LIN {X 0,Y 195.024,Z 1205.929,A -85,B 0,C 180,E1 26196.812,E2 26196.812} C_VEL
LIN {X 0,Y 201.887,Z 1195.668,A -85,B 0,C 180,E1 26216.922,E2 26216.922} C_VEL
LIN {X 0,Y 228.615,Z 1170.249,A -85,B 0,C 180,E1 26237.028,E2 26237.028} C_VEL
LIN {X 0,Y 271.892,Z 1129.75,A -85,B 0,C 180,E1 26251.738,E2 26251.738} C_VEL
LIN {X 0,Y 319.813,Z 1076.72,A -85,B 0,C 180,E1 26261.083,E2 26261.083} C_VEL
LIN {X 0,Y 361.01,Z 1018.168,A -85,B 0,C 180,E1 26266.67,E2 26266.67} C_VEL
LIN {X 0,Y 361.601,Z 999.754,A -85,B 0,C 180,E1 26275.219,E2 26275.219} C_VEL
LIN {X 0,Y 361.684,Z 993.07,A -85,B 0,C 180,E1 26283.639,E2 26283.639} C_VEL
LIN {X 0,Y 360.895,Z 1000.649,A -85,B 0,C 180,E1 26292.409,E2 26292.409} C_VEL
LIN {X 0,Y 359.633,Z 1018.396,A -85,B 0,C 180,E1 26300.562,E2 26300.562} C_VEL
LIN {X 0,Y 315.236,Z 1080.357,A -85,B 0,C 180,E1 26306.923,E2 26306.923} C_VEL
LIN {X 0,Y 267.258,Z 1131.688,A -85,B 0,C 180,E1 26316.736,E2 26316.736} C_VEL
LIN {X 0,Y 264.551,Z 1134.275,A -85,B 0,C 180,E1 26317.455,E2 26317.455} C_VEL
LIN {X 0,Y 240.513,Z 1151.989,A -85,B 0,C 180,E1 26321.828,E2 26321.828} C_VEL
LIN {X 0,Y 204.312,Z 1182.961,A -85,B 0,C 180,E1 26339.909,E2 26339.909} C_VEL
LIN {X 0,Y 188.932,Z 1198.697,A -85,B 0,C 180,E1 26360.642,E2 26360.642} C_VEL
LIN {X 0,Y 186.458,Z 1202.773,A -85,B 0,C 180,E1 26376.895,E2 26376.895} C_VEL
LIN {X 0,Y 189.671,Z 1199.838,A -85,B 0,C 180,E1 26395.976,E2 26395.976} C_VEL
LIN {X 0,Y 209.352,Z 1185.393,A -85,B 0,C 180,E1 26417.213,E2 26417.213} C_VEL
LIN {X 0,Y 251.624,Z 1155.697,A -85,B 0,C 180,E1 26434.833,E2 26434.833} C_VEL
LIN {X 0,Y 304.449,Z 1112.39,A -85,B 0,C 180,E1 26446.069,E2 26446.069} C_VEL
LIN {X 0,Y 355.93,Z 1058.355,A -85,B 0,C 180,E1 26452.911,E2 26452.911} C_VEL
LIN {X 0,Y 371.692,Z 1038.15,A -85,B 0,C 180,E1 26454.701,E2 26454.701} C_VEL
LIN {X 0,Y 373.231,Z 1031.62,A -85,B 0,C 180,E1 26461.134,E2 26461.134} C_VEL
LIN {X 0,Y 372.915,Z 1033.797,A -85,B 0,C 180,E1 26468.154,E2 26468.154} C_VEL
LIN {X 0,Y 370.664,Z 1040.666,A -85,B 0,C 180,E1 26472.243,E2 26472.243} C_VEL
LIN {X 0,Y 321.62,Z 1097.337,A -85,B 0,C 180,E1 26477.917,E2 26477.917} C_VEL
LIN {X 0,Y 267.836,Z 1145.357,A -85,B 0,C 180,E1 26487.532,E2 26487.532} C_VEL
LIN {X 0,Y 221.377,Z 1179.857,A -85,B 0,C 180,E1 26502.685,E2 26502.685} C_VEL
LIN {X 0,Y 192.93,Z 1200.687,A -85,B 0,C 180,E1 26524.578,E2 26524.578} C_VEL
LIN {X 0,Y 187.059,Z 1206.716,A -85,B 0,C 180,E1 26543.127,E2 26543.127} C_VEL
LIN {X 0,Y 187.015,Z 1205.813,A -85,B 0,C 180,E1 26557.105,E2 26557.105} C_VEL
LIN {X 0,Y 194.537,Z 1195.482,A -85,B 0,C 180,E1 26578.027,E2 26578.027} C_VEL
LIN {X 0,Y 223.002,Z 1169.972,A -85,B 0,C 180,E1 26598.599,E2 26598.599} C_VEL
LIN {X 0,Y 268.014,Z 1129.339,A -85,B 0,C 180,E1 26613.321,E2 26613.321} C_VEL
LIN {X 0,Y 316.678,Z 1076.788,A -85,B 0,C 180,E1 26622.446,E2 26622.446} C_VEL
LIN {X 0,Y 356.066,Z 1022.174,A -85,B 0,C 180,E1 26627.651,E2 26627.651} C_VEL
LIN {X 0,Y 357.113,Z 1004.901,A -85,B 0,C 180,E1 26636.379,E2 26636.379} C_VEL
LIN {X 0,Y 357.474,Z 999.9,A -85,B 0,C 180,E1 26643.682,E2 26643.682} C_VEL
LIN {X 0,Y 356.208,Z 1008.216,A -85,B 0,C 180,E1 26652.952,E2 26652.952} C_VEL
LIN {X 0,Y 353.927,Z 1024.296,A -85,B 0,C 180,E1 26659.943,E2 26659.943} C_VEL
LIN {X 0,Y 308.648,Z 1084.424,A -85,B 0,C 180,E1 26666.084,E2 26666.084} C_VEL
LIN {X 0,Y 259.49,Z 1134.902,A -85,B 0,C 180,E1 26676.09,E2 26676.09} C_VEL
LIN {X 0,Y 240.513,Z 1151.989,A -85,B 0,C 180,E1 26681.828,E2 26681.828} C_VEL
LIN {X 0,Y 216.948,Z 1167.301,A -85,B 0,C 180,E1 26687.305,E2 26687.305} C_VEL
LIN {X 0,Y 187.065,Z 1192.104,A -85,B 0,C 180,E1 26708.47,E2 26708.47} C_VEL
LIN {X 0,Y 179.568,Z 1201.352,A -85,B 0,C 180,E1 26727.459,E2 26727.459} C_VEL
LIN {X 0,Y 178.358,Z 1202.913,A -85,B 0,C 180,E1 26742.156,E2 26742.156} C_VEL
LIN {X 0,Y 186.636,Z 1196.622,A -85,B 0,C 180,E1 26764.382,E2 26764.382} C_VEL
LIN {X 0,Y 218.438,Z 1175.736,A -85,B 0,C 180,E1 26786.538,E2 26786.538} C_VEL
LIN {X 0,Y 267.906,Z 1140.876,A -85,B 0,C 180,E1 26801.382,E2 26801.382} C_VEL
LIN {X 0,Y 323.344,Z 1092.416,A -85,B 0,C 180,E1 26810.602,E2 26810.602} C_VEL
LIN {X 0,Y 366.777,Z 1043.151,A -85,B 0,C 180,E1 26815.553,E2 26815.553} C_VEL
LIN {X 0,Y 368.312,Z 1037.517,A -85,B 0,C 180,E1 26823.511,E2 26823.511} C_VEL
LIN {X 0,Y 366.986,Z 1043.658,A -85,B 0,C 180,E1 26831.058,E2 26831.058} C_VEL
LIN {X 0,Y 314.684,Z 1102.026,A -85,B 0,C 180,E1 26837.109,E2 26837.109} C_VEL
LIN {X 0,Y 259.292,Z 1149.207,A -85,B 0,C 180,E1 26847.01,E2 26847.01} C_VEL
LIN {X 0,Y 210.752,Z 1183.326,A -85,B 0,C 180,E1 26863.433,E2 26863.433} C_VEL
LIN {X 0,Y 183.93,Z 1201.951,A -85,B 0,C 180,E1 26885.994,E2 26885.994} C_VEL
LIN {X 0,Y 178.992,Z 1206.922,A -85,B 0,C 180,E1 26907.691,E2 26907.691} C_VEL
LIN {X 0,Y 180.833,Z 1202.479,A -85,B 0,C 180,E1 26927.202,E2 26927.202} C_VEL
LIN {X 0,Y 197.975,Z 1185.627,A -85,B 0,C 180,E1 26949.358,E2 26949.358} C_VEL
LIN {X 0,Y 236.545,Z 1153.621,A -85,B 0,C 180,E1 26967.534,E2 26967.534} C_VEL
LIN {X 0,Y 286.12,Z 1107.52,A -85,B 0,C 180,E1 26979.377,E2 26979.377} C_VEL
LIN {X 0,Y 335.559,Z 1049.133,A -85,B 0,C 180,E1 26986.721,E2 26986.721} C_VEL
LIN {X 0,Y 351.217,Z 1025.839,A -85,B 0,C 180,E1 26988.826,E2 26988.826} C_VEL
LIN {X 0,Y 352.633,Z 1010,A -85,B 0,C 180,E1 26997.721,E2 26997.721} C_VEL
LIN {X 0,Y 352.974,Z 1006.543,A -85,B 0,C 180,E1 27003.729,E2 27003.729} C_VEL
LIN {X 0,Y 351.613,Z 1014.433,A -85,B 0,C 180,E1 27012.617,E2 27012.617} C_VEL
LIN {X 0,Y 349.457,Z 1027.85,A -85,B 0,C 180,E1 27018.921,E2 27018.921} C_VEL
LIN {X 0,Y 303.375,Z 1087.058,A -85,B 0,C 180,E1 27025.006,E2 27025.006} C_VEL
LIN {X 0,Y 253.893,Z 1136.158,A -85,B 0,C 180,E1 27034.849,E2 27034.849} C_VEL
LIN {X 0,Y 216.948,Z 1167.301,A -85,B 0,C 180,E1 27047.305,E2 27047.305} C_VEL
LIN {X 0,Y 194.903,Z 1179.91,A -85,B 0,C 180,E1 27054.219,E2 27054.219} C_VEL
LIN {X 0,Y 174.022,Z 1197.858,A -85,B 0,C 180,E1 27077.284,E2 27077.284} C_VEL
LIN {X 0,Y 170.807,Z 1202.507,A -85,B 0,C 180,E1 27092.42,E2 27092.42} C_VEL
LIN {X 0,Y 172.398,Z 1201.52,A -85,B 0,C 180,E1 27113.196,E2 27113.196} C_VEL
LIN {X 0,Y 190.131,Z 1190.023,A -85,B 0,C 180,E1 27135.745,E2 27135.745} C_VEL
LIN {X 0,Y 232.547,Z 1163.511,A -85,B 0,C 180,E1 27155.129,E2 27155.129} C_VEL
LIN {X 0,Y 287.445,Z 1123.09,A -85,B 0,C 180,E1 27167.218,E2 27167.218} C_VEL
LIN {X 0,Y 342.611,Z 1070.565,A -85,B 0,C 180,E1 27174.462,E2 27174.462} C_VEL
LIN {X 0,Y 361.922,Z 1047.935,A -85,B 0,C 180,E1 27176.703,E2 27176.703} C_VEL
LIN {X 0,Y 363.229,Z 1043.712,A -85,B 0,C 180,E1 27183.56,E2 27183.56} C_VEL
LIN {X 0,Y 361.999,Z 1048.851,A -85,B 0,C 180,E1 27190.283,E2 27190.283} C_VEL
LIN {X 0,Y 309.639,Z 1104.957,A -85,B 0,C 180,E1 27196.025,E2 27196.025} C_VEL
LIN {X 0,Y 252.779,Z 1151.524,A -85,B 0,C 180,E1 27205.989,E2 27205.989} C_VEL
LIN {X 0,Y 203.201,Z 1184.583,A -85,B 0,C 180,E1 27222.666,E2 27222.666} C_VEL
LIN {X 0,Y 176.98,Z 1201.491,A -85,B 0,C 180,E1 27244.009,E2 27244.009} C_VEL
LIN {X 0,Y 171.056,Z 1206.558,A -85,B 0,C 180,E1 27262.48,E2 27262.48} C_VEL
LIN {X 0,Y 171.033,Z 1205.58,A -85,B 0,C 180,E1 27277.773,E2 27277.773} C_VEL
LIN {X 0,Y 180.096,Z 1195.09,A -85,B 0,C 180,E1 27300.502,E2 27300.502} C_VEL
LIN {X 0,Y 211.654,Z 1169.878,A -85,B 0,C 180,E1 27321.738,E2 27321.738} C_VEL
LIN {X 0,Y 259.327,Z 1129.967,A -85,B 0,C 180,E1 27336.295,E2 27336.295} C_VEL
LIN {X 0,Y 310.115,Z 1077.93,A -85,B 0,C 180,E1 27345.135,E2 27345.135} C_VEL
LIN {X 0,Y 346.289,Z 1030.608,A -85,B 0,C 180,E1 27349.612,E2 27349.612} C_VEL
LIN {X 0,Y 348.03,Z 1016.909,A -85,B 0,C 180,E1 27357.535,E2 27357.535} C_VEL
LIN {X 0,Y 348.449,Z 1013.197,A -85,B 0,C 180,E1 27363.777,E2 27363.777} C_VEL
LIN {X 0,Y 346.636,Z 1021.689,A -85,B 0,C 180,E1 27373.027,E2 27373.027} C_VEL
LIN {X 0,Y 344.666,Z 1032.036,A -85,B 0,C 180,E1 27377.912,E2 27377.912} C_VEL
LIN {X 0,Y 296.035,Z 1092.078,A -85,B 0,C 180,E1 27384.245,E2 27384.245} C_VEL
LIN {X 0,Y 244.515,Z 1140.715,A -85,B 0,C 180,E1 27394.541,E2 27394.541} C_VEL
LIN {X 0,Y 199.997,Z 1175.914,A -85,B 0,C 180,E1 27411.115,E2 27411.115} C_VEL
LIN {X 0,Y 194.903,Z 1179.91,A -85,B 0,C 180,E1 27414.219,E2 27414.219} C_VEL
LIN {X 0,Y 175.399,Z 1189.873,A -85,B 0,C 180,E1 27422.94,E2 27422.94} C_VEL
LIN {X 0,Y 163.601,Z 1201.601,A -85,B 0,C 180,E1 27447.211,E2 27447.211} C_VEL
LIN {X 0,Y 162.366,Z 1203.067,A -85,B 0,C 180,E1 27463.375,E2 27463.375} C_VEL
LIN {X 0,Y 170.733,Z 1197.771,A -85,B 0,C 180,E1 27485.131,E2 27485.131} C_VEL
LIN {X 0,Y 204.225,Z 1178.439,A -85,B 0,C 180,E1 27508.49,E2 27508.49} C_VEL
LIN {X 0,Y 257.447,Z 1144.23,A -85,B 0,C 180,E1 27523.933,E2 27523.933} C_VEL
LIN {X 0,Y 314.998,Z 1097.224,A -85,B 0,C 180,E1 27532.941,E2 27532.941} C_VEL
LIN {X 0,Y 356.585,Z 1053.458,A -85,B 0,C 180,E1 27537.284,E2 27537.284} C_VEL
LIN {X 0,Y 358.084,Z 1049.889,A -85,B 0,C 180,E1 27543.611,E2 27543.611} C_VEL
LIN {X 0,Y 356.477,Z 1054.209,A -85,B 0,C 180,E1 27549.367,E2 27549.367} C_VEL
LIN {X 0,Y 302.291,Z 1109.824,A -85,B 0,C 180,E1 27555.214,E2 27555.214} C_VEL
LIN {X 0,Y 246.344,Z 1153.614,A -85,B 0,C 180,E1 27564.912,E2 27564.912} C_VEL
LIN {X 0,Y 196.648,Z 1185.176,A -85,B 0,C 180,E1 27581.356,E2 27581.356} C_VEL
LIN {X 0,Y 167.605,Z 1202.876,A -85,B 0,C 180,E1 27606.1,E2 27606.1} C_VEL
LIN {X 0,Y 162.977,Z 1206.728,A -85,B 0,C 180,E1 27627.464,E2 27627.464} C_VEL
LIN {X 0,Y 163.808,Z 1203.967,A -85,B 0,C 180,E1 27643.799,E2 27643.799} C_VEL
LIN {X 0,Y 178.375,Z 1190.651,A -85,B 0,C 180,E1 27667.123,E2 27667.123} C_VEL
LIN {X 0,Y 216.464,Z 1161.923,A -85,B 0,C 180,E1 27687.442,E2 27687.442} C_VEL
LIN {X 0,Y 267.953,Z 1118.788,A -85,B 0,C 180,E1 27700.373,E2 27700.373} C_VEL
LIN {X 0,Y 320.137,Z 1063.085,A -85,B 0,C 180,E1 27708.147,E2 27708.147} C_VEL
LIN {X 0,Y 341.461,Z 1034.746,A -85,B 0,C 180,E1 27710.703,E2 27710.703} C_VEL
LIN {X 0,Y 343.382,Z 1022.137,A -85,B 0,C 180,E1 27718.768,E2 27718.768} C_VEL
LIN {X 0,Y 343.3,Z 1020.817,A -85,B 0,C 180,E1 27726.376,E2 27726.376} C_VEL
LIN {X 0,Y 340.899,Z 1032.315,A -85,B 0,C 180,E1 27735.232,E2 27735.232} C_VEL
LIN {X 0,Y 338.436,Z 1037.977,A -85,B 0,C 180,E1 27737.036,E2 27737.036} C_VEL
LIN {X 0,Y 289.523,Z 1095.934,A -85,B 0,C 180,E1 27743.308,E2 27743.308} C_VEL
LIN {X 0,Y 237.342,Z 1143.233,A -85,B 0,C 180,E1 27753.63,E2 27753.63} C_VEL
LIN {X 0,Y 191.916,Z 1177.502,A -85,B 0,C 180,E1 27770.623,E2 27770.623} C_VEL
LIN {X 0,Y 175.399,Z 1189.873,A -85,B 0,C 180,E1 27782.94,E2 27782.94} C_VEL
LIN {X 0,Y 159.541,Z 1197.139,A -85,B 0,C 180,E1 27793.572,E2 27793.572} C_VEL
LIN {X 0,Y 154.715,Z 1202.757,A -85,B 0,C 180,E1 27812.672,E2 27812.672} C_VEL
LIN {X 0,Y 157.122,Z 1201.626,A -85,B 0,C 180,E1 27835.605,E2 27835.605} C_VEL
LIN {X 0,Y 179.789,Z 1189.181,A -85,B 0,C 180,E1 27860.66,E2 27860.66} C_VEL
LIN {X 0,Y 226.507,Z 1162.681,A -85,B 0,C 180,E1 27879.414,E2 27879.414} C_VEL
LIN {X 0,Y 285.565,Z 1121.357,A -85,B 0,C 180,E1 27890.85,E2 27890.85} C_VEL
LIN {X 0,Y 342.838,Z 1068.116,A -85,B 0,C 180,E1 27897.465,E2 27897.465} C_VEL
LIN {X 0,Y 351.621,Z 1058.278,A -85,B 0,C 180,E1 27898.39,E2 27898.39} C_VEL
LIN {X 0,Y 352.722,Z 1055.854,A -85,B 0,C 180,E1 27903.666,E2 27903.666} C_VEL
LIN {X 0,Y 350.645,Z 1059.989,A -85,B 0,C 180,E1 27908.45,E2 27908.45} C_VEL
LIN {X 0,Y 295.21,Z 1114.413,A -85,B 0,C 180,E1 27914.341,E2 27914.341} C_VEL
LIN {X 0,Y 236.203,Z 1158.188,A -85,B 0,C 180,E1 27924.62,E2 27924.62} C_VEL
LIN {X 0,Y 185.023,Z 1188.672,A -85,B 0,C 180,E1 27942.607,E2 27942.607} C_VEL
LIN {X 0,Y 160.106,Z 1202.836,A -85,B 0,C 180,E1 27964.905,E2 27964.905} C_VEL
LIN {X 0,Y 154.957,Z 1206.63,A -85,B 0,C 180,E1 27987.332,E2 27987.332} C_VEL
LIN {X 0,Y 155.892,Z 1203.919,A -85,B 0,C 180,E1 28004.224,E2 28004.224} C_VEL
LIN {X 0,Y 172.808,Z 1189.67,A -85,B 0,C 180,E1 28029.697,E2 28029.697} C_VEL
LIN {X 0,Y 214.474,Z 1159.782,A -85,B 0,C 180,E1 28050.165,E2 28050.165} C_VEL
LIN {X 0,Y 267.017,Z 1116.65,A -85,B 0,C 180,E1 28062.399,E2 28062.399} C_VEL
LIN {X 0,Y 319.726,Z 1060.934,A -85,B 0,C 180,E1 28069.771,E2 28069.771} C_VEL
LIN {X 0,Y 336.527,Z 1038.815,A -85,B 0,C 180,E1 28071.851,E2 28071.851} C_VEL
LIN {X 0,Y 338.699,Z 1027.59,A -85,B 0,C 180,E1 28080.034,E2 28080.034} C_VEL
LIN {X 0,Y 338.448,Z 1027.327,A -85,B 0,C 180,E1 28086.468,E2 28086.468} C_VEL
LIN {X 0,Y 335.695,Z 1038.142,A -85,B 0,C 180,E1 28094.928,E2 28094.928} C_VEL
LIN {X 0,Y 332.593,Z 1043.487,A -85,B 0,C 180,E1 28096.1,E2 28096.1} C_VEL
LIN {X 0,Y 281.703,Z 1101.168,A -85,B 0,C 180,E1 28102.528,E2 28102.528} C_VEL
LIN {X 0,Y 227.604,Z 1147.871,A -85,B 0,C 180,E1 28113.392,E2 28113.392} C_VEL
LIN {X 0,Y 182.053,Z 1180.397,A -85,B 0,C 180,E1 28131.162,E2 28131.162} C_VEL
LIN {X 0,Y 159.541,Z 1197.139,A -85,B 0,C 180,E1 28153.572,E2 28153.572} C_VEL
LIN {X 0,Y 147.667,Z 1201.624,A -85,B 0,C 180,E1 28166.029,E2 28166.029} C_VEL
LIN {X 0,Y 146.425,Z 1203.221,A -85,B 0,C 180,E1 28184.862,E2 28184.862} C_VEL
LIN {X 0,Y 158.718,Z 1196.977,A -85,B 0,C 180,E1 28210.575,E2 28210.575} C_VEL
LIN {X 0,Y 199.919,Z 1176.032,A -85,B 0,C 180,E1 28234.358,E2 28234.358} C_VEL
LIN {X 0,Y 257.121,Z 1141.164,A -85,B 0,C 180,E1 28248.403,E2 28248.403} C_VEL
LIN {X 0,Y 316.922,Z 1093.295,A -85,B 0,C 180,E1 28256.437,E2 28256.437} C_VEL
LIN {X 0,Y 346.542,Z 1063.427,A -85,B 0,C 180,E1 28259.391,E2 28259.391} C_VEL
LIN {X 0,Y 346.925,Z 1062.937,A -85,B 0,C 180,E1 28266.243,E2 28266.243} C_VEL
LIN {X 0,Y 345.823,Z 1064.684,A -85,B 0,C 180,E1 28267.446,E2 28267.446} C_VEL
LIN {X 0,Y 288.195,Z 1118.947,A -85,B 0,C 180,E1 28273.424,E2 28273.424} C_VEL
LIN {X 0,Y 226.599,Z 1162.221,A -85,B 0,C 180,E1 28284.171,E2 28284.171} C_VEL
LIN {X 0,Y 175.411,Z 1190.811,A -85,B 0,C 180,E1 28302.853,E2 28302.853} C_VEL
LIN {X 0,Y 149.739,Z 1204.545,A -85,B 0,C 180,E1 28329.381,E2 28329.381} C_VEL
LIN {X 0,Y 146.935,Z 1206.532,A -85,B 0,C 180,E1 28347.186,E2 28347.186} C_VEL
LIN {X 0,Y 148.02,Z 1203.78,A -85,B 0,C 180,E1 28364.998,E2 28364.998} C_VEL
LIN {X 0,Y 166.423,Z 1189.44,A -85,B 0,C 180,E1 28391.546,E2 28391.546} C_VEL
LIN {X 0,Y 209.967,Z 1159.747,A -85,B 0,C 180,E1 28412.053,E2 28412.053} C_VEL
LIN {X 0,Y 264.373,Z 1116.392,A -85,B 0,C 180,E1 28424.105,E2 28424.105} C_VEL
LIN {X 0,Y 318.032,Z 1060.687,A -85,B 0,C 180,E1 28431.225,E2 28431.225} C_VEL
LIN {X 0,Y 331.562,Z 1043.442,A -85,B 0,C 180,E1 28432.766,E2 28432.766} C_VEL
LIN {X 0,Y 334.187,Z 1033.039,A -85,B 0,C 180,E1 28441.335,E2 28441.335} C_VEL
LIN {X 0,Y 332.728,Z 1036.085,A -85,B 0,C 180,E1 28449.217,E2 28449.217} C_VEL
LIN {X 0,Y 329.231,Z 1045.83,A -85,B 0,C 180,E1 28454.895,E2 28454.895} C_VEL
LIN {X 0,Y 276.505,Z 1103.865,A -85,B 0,C 180,E1 28461.322,E2 28461.322} C_VEL
LIN {X 0,Y 221.869,Z 1149.316,A -85,B 0,C 180,E1 28472.009,E2 28472.009} C_VEL
LIN {X 0,Y 173.982,Z 1181.882,A -85,B 0,C 180,E1 28490.624,E2 28490.624} C_VEL
LIN {X 0,Y 150.614,Z 1198.38,A -85,B 0,C 180,E1 28515.266,E2 28515.266} C_VEL
LIN {X 0,Y 147.667,Z 1201.624,A -85,B 0,C 180,E1 28526.029,E2 28526.029} C_VEL
LIN {X 0,Y 138.179,Z 1203.374,A -85,B 0,C 180,E1 28539.823,E2 28539.823} C_VEL
LIN {X 0,Y 145.716,Z 1200.006,A -85,B 0,C 180,E1 28564.759,E2 28564.759} C_VEL
LIN {X 0,Y 181.432,Z 1183.29,A -85,B 0,C 180,E1 28591.167,E2 28591.167} C_VEL
LIN {X 0,Y 237.938,Z 1152.249,A -85,B 0,C 180,E1 28607.263,E2 28607.263} C_VEL
LIN {X 0,Y 299.396,Z 1107.866,A -85,B 0,C 180,E1 28616.216,E2 28616.216} C_VEL
LIN {X 0,Y 341.014,Z 1068.791,A -85,B 0,C 180,E1 28620.197,E2 28620.197} C_VEL
LIN {X 0,Y 341.286,Z 1068.795,A -85,B 0,C 180,E1 28626.346,E2 28626.346} C_VEL
LIN {X 0,Y 282.135,Z 1122.433,A -85,B 0,C 180,E1 28632.331,E2 28632.331} C_VEL
LIN {X 0,Y 221.5,Z 1163.382,A -85,B 0,C 180,E1 28642.623,E2 28642.623} C_VEL
LIN {X 0,Y 167.411,Z 1191.989,A -85,B 0,C 180,E1 28662.183,E2 28662.183} C_VEL
LIN {X 0,Y 142.101,Z 1204.505,A -85,B 0,C 180,E1 28688.218,E2 28688.218} C_VEL
LIN {X 0,Y 138.927,Z 1206.435,A -85,B 0,C 180,E1 28707.024,E2 28707.024} C_VEL
LIN {X 0,Y 140.166,Z 1203.641,A -85,B 0,C 180,E1 28725.86,E2 28725.86} C_VEL
LIN {X 0,Y 160.229,Z 1189.208,A -85,B 0,C 180,E1 28753.54,E2 28753.54} C_VEL
LIN {X 0,Y 205.487,Z 1159.882,A -85,B 0,C 180,E1 28773.936,E2 28773.936} C_VEL
LIN {X 0,Y 261.93,Z 1116.144,A -85,B 0,C 180,E1 28785.851,E2 28785.851} C_VEL
LIN {X 0,Y 316.255,Z 1060.785,A -85,B 0,C 180,E1 28792.667,E2 28792.667} C_VEL
LIN {X 0,Y 326.784,Z 1047.553,A -85,B 0,C 180,E1 28794.041,E2 28794.041} C_VEL
LIN {X 0,Y 329.097,Z 1039.254,A -85,B 0,C 180,E1 28801.355,E2 28801.355} C_VEL
LIN {X 0,Y 327.488,Z 1042.536,A -85,B 0,C 180,E1 28809.365,E2 28809.365} C_VEL
LIN {X 0,Y 325.326,Z 1048.992,A -85,B 0,C 180,E1 28813.715,E2 28813.715} C_VEL
LIN {X 0,Y 271.63,Z 1106.202,A -85,B 0,C 180,E1 28820.036,E2 28820.036} C_VEL
LIN {X 0,Y 216.265,Z 1150.637,A -85,B 0,C 180,E1 28830.553,E2 28830.553} C_VEL
LIN {X 0,Y 167.771,Z 1182.132,A -85,B 0,C 180,E1 28848.86,E2 28848.86} C_VEL
LIN {X 0,Y 142.872,Z 1198.552,A -85,B 0,C 180,E1 28874.448,E2 28874.448} C_VEL
LIN {X 0,Y 138.611,Z 1203.005,A -85,B 0,C 180,E1 28892.983,E2 28892.983} C_VEL
LIN {X 0,Y 138.179,Z 1203.374,A -85,B 0,C 180,E1 28899.823,E2 28899.823} C_VEL
LIN {X 0,Y 132.417,Z 1202.621,A -85,B 0,C 180,E1 28914.71,E2 28914.71} C_VEL
LIN {X 0,Y 154.414,Z 1193.424,A -85,B 0,C 180,E1 28941.642,E2 28941.642} C_VEL
LIN {X 0,Y 205.954,Z 1169.136,A -85,B 0,C 180,E1 28962.803,E2 28962.803} C_VEL
LIN {X 0,Y 268.861,Z 1130.635,A -85,B 0,C 180,E1 28974.343,E2 28974.343} C_VEL
LIN {X 0,Y 329.558,Z 1080.107,A -85,B 0,C 180,E1 28980.698,E2 28980.698} C_VEL
LIN {X 0,Y 335.924,Z 1073.712,A -85,B 0,C 180,E1 28981.26,E2 28981.26} C_VEL
LIN {X 0,Y 335.811,Z 1073.988,A -85,B 0,C 180,E1 28985.209,E2 28985.209} C_VEL
LIN {X 0,Y 274.537,Z 1127.175,A -85,B 0,C 180,E1 28991.403,E2 28991.403} C_VEL
LIN {X 0,Y 212.331,Z 1166.952,A -85,B 0,C 180,E1 29001.999,E2 29001.999} C_VEL
LIN {X 0,Y 159.904,Z 1192.938,A -85,B 0,C 180,E1 29021.141,E2 29021.141} C_VEL
LIN {X 0,Y 134.557,Z 1204.464,A -85,B 0,C 180,E1 29046.928,E2 29046.928} C_VEL
LIN {X 0,Y 130.903,Z 1206.337,A -85,B 0,C 180,E1 29066.842,E2 29066.842} C_VEL
LIN {X 0,Y 132.371,Z 1203.502,A -85,B 0,C 180,E1 29086.821,E2 29086.821} C_VEL
LIN {X 0,Y 154.223,Z 1188.975,A -85,B 0,C 180,E1 29115.7,E2 29115.7} C_VEL
LIN {X 0,Y 202.202,Z 1159.345,A -85,B 0,C 180,E1 29136.172,E2 29136.172} C_VEL
LIN {X 0,Y 259.272,Z 1116.302,A -85,B 0,C 180,E1 29147.564,E2 29147.564} C_VEL
LIN {X 0,Y 314.983,Z 1060.526,A -85,B 0,C 180,E1 29154.151,E2 29154.151} C_VEL
LIN {X 0,Y 321.814,Z 1052.135,A -85,B 0,C 180,E1 29155.056,E2 29155.056} C_VEL
LIN {X 0,Y 323.975,Z 1045.478,A -85,B 0,C 180,E1 29161.377,E2 29161.377} C_VEL
LIN {X 0,Y 322.215,Z 1048.985,A -85,B 0,C 180,E1 29169.52,E2 29169.52} C_VEL
LIN {X 0,Y 319.254,Z 1054.681,A -85,B 0,C 180,E1 29172.724,E2 29172.724} C_VEL
LIN {X 0,Y 263.465,Z 1111.48,A -85,B 0,C 180,E1 29179.189,E2 29179.189} C_VEL
LIN {X 0,Y 206.525,Z 1154.812,A -85,B 0,C 180,E1 29190.112,E2 29190.112} C_VEL
LIN {X 0,Y 157.884,Z 1184.623,A -85,B 0,C 180,E1 29209.379,E2 29209.379} C_VEL
LIN {X 0,Y 135.141,Z 1198.725,A -85,B 0,C 180,E1 29233.534,E2 29233.534} C_VEL
LIN {X 0,Y 130.553,Z 1203.12,A -85,B 0,C 180,E1 29253.167,E2 29253.167} C_VEL
LIN {X 0,Y 132.417,Z 1202.621,A -85,B 0,C 180,E1 29274.71,E2 29274.71} C_VEL
LIN {X 0,Y 132.879,Z 1199.72,A -85,B 0,C 180,E1 29290.028,E2 29290.028} C_VEL
LIN {X 0,Y 176.359,Z 1182.039,A -85,B 0,C 180,E1 29317.158,E2 29317.158} C_VEL
LIN {X 0,Y 239.126,Z 1149.306,A -85,B 0,C 180,E1 29332.094,E2 29332.094} C_VEL
LIN {X 0,Y 302.153,Z 1104.493,A -85,B 0,C 180,E1 29339.842,E2 29339.842} C_VEL
LIN {X 0,Y 330.295,Z 1079.221,A -85,B 0,C 180,E1 29342.382,E2 29342.382} C_VEL
LIN {X 0,Y 329.781,Z 1079.81,A -85,B 0,C 180,E1 29344.378,E2 29344.378} C_VEL
LIN {X 0,Y 267.617,Z 1131.321,A -85,B 0,C 180,E1 29350.362,E2 29350.362} C_VEL
LIN {X 0,Y 203.187,Z 1170.337,A -85,B 0,C 180,E1 29361.317,E2 29361.317} C_VEL
LIN {X 0,Y 150.603,Z 1194.711,A -85,B 0,C 180,E1 29381.139,E2 29381.139} C_VEL
LIN {X 0,Y 124.451,Z 1205.481,A -85,B 0,C 180,E1 29412.435,E2 29412.435} C_VEL
LIN {X 0,Y 122.824,Z 1205.9,A -85,B 0,C 180,E1 29433.716,E2 29433.716} C_VEL
LIN {X 0,Y 131.054,Z 1198.853,A -85,B 0,C 180,E1 29461.59,E2 29461.59} C_VEL
LIN {X 0,Y 169.182,Z 1177.176,A -85,B 0,C 180,E1 29488.671,E2 29488.671} C_VEL
LIN {X 0,Y 226.764,Z 1140.03,A -85,B 0,C 180,E1 29504.466,E2 29504.466} C_VEL
LIN {X 0,Y 285.221,Z 1090.774,A -85,B 0,C 180,E1 29512.79,E2 29512.79} C_VEL
LIN {X 0,Y 316.664,Z 1057.016,A -85,B 0,C 180,E1 29515.916,E2 29515.916} C_VEL
LIN {X 0,Y 318.741,Z 1051.593,A -85,B 0,C 180,E1 29521.399,E2 29521.399} C_VEL
LIN {X 0,Y 317.435,Z 1053.495,A -85,B 0,C 180,E1 29527.968,E2 29527.968} C_VEL
LIN {X 0,Y 314.902,Z 1058.474,A -85,B 0,C 180,E1 29531.555,E2 29531.555} C_VEL
LIN {X 0,Y 259.267,Z 1113.389,A -85,B 0,C 180,E1 29537.746,E2 29537.746} C_VEL
LIN {X 0,Y 199.681,Z 1157.076,A -85,B 0,C 180,E1 29548.873,E2 29548.873} C_VEL
LIN {X 0,Y 149.877,Z 1185.993,A -85,B 0,C 180,E1 29568.661,E2 29568.661} C_VEL
LIN {X 0,Y 125.017,Z 1200.781,A -85,B 0,C 180,E1 29599.337,E2 29599.337} C_VEL
LIN {X 0,Y 122.155,Z 1203.583,A -85,B 0,C 180,E1 29620.559,E2 29620.559} C_VEL
LIN {X 0,Y 132.879,Z 1199.72,A -85,B 0,C 180,E1 29650.028,E2 29650.028} C_VEL
LIN {X 0,Y 140.276,Z 1194.818,A -85,B 0,C 180,E1 29664.492,E2 29664.492} C_VEL
LIN {X 0,Y 197.177,Z 1170.92,A -85,B 0,C 180,E1 29686.588,E2 29686.588} C_VEL
LIN {X 0,Y 263.401,Z 1133.001,A -85,B 0,C 180,E1 29697.544,E2 29697.544} C_VEL
LIN {X 0,Y 324.124,Z 1084.943,A -85,B 0,C 180,E1 29703.317,E2 29703.317} C_VEL
LIN {X 0,Y 260.948,Z 1135.103,A -85,B 0,C 180,E1 29709.241,E2 29709.241} C_VEL
LIN {X 0,Y 194.165,Z 1173.425,A -85,B 0,C 180,E1 29720.521,E2 29720.521} C_VEL
LIN {X 0,Y 140.978,Z 1196.285,A -85,B 0,C 180,E1 29741.347,E2 29741.347} C_VEL
LIN {X 0,Y 116.709,Z 1205.422,A -85,B 0,C 180,E1 29771.228,E2 29771.228} C_VEL
LIN {X 0,Y 114.801,Z 1205.795,A -85,B 0,C 180,E1 29793.976,E2 29793.976} C_VEL
LIN {X 0,Y 124.085,Z 1198.67,A -85,B 0,C 180,E1 29823.591,E2 29823.591} C_VEL
LIN {X 0,Y 164.995,Z 1176.916,A -85,B 0,C 180,E1 29851.149,E2 29851.149} C_VEL
LIN {X 0,Y 224.338,Z 1139.862,A -85,B 0,C 180,E1 29866.483,E2 29866.483} C_VEL
LIN {X 0,Y 284.179,Z 1090.349,A -85,B 0,C 180,E1 29874.45,E2 29874.45} C_VEL
LIN {X 0,Y 311.764,Z 1061.343,A -85,B 0,C 180,E1 29877.288,E2 29877.288} C_VEL
LIN {X 0,Y 313.314,Z 1057.261,A -85,B 0,C 180,E1 29884.201,E2 29884.201} C_VEL
LIN {X 0,Y 309.921,Z 1063.143,A -85,B 0,C 180,E1 29890.424,E2 29890.424} C_VEL
LIN {X 0,Y 251.866,Z 1118.072,A -85,B 0,C 180,E1 29896.702,E2 29896.702} C_VEL
LIN {X 0,Y 191.991,Z 1159.837,A -85,B 0,C 180,E1 29907.787,E2 29907.787} C_VEL
LIN {X 0,Y 139.863,Z 1188.326,A -85,B 0,C 180,E1 29929.197,E2 29929.197} C_VEL
LIN {X 0,Y 117.141,Z 1200.928,A -85,B 0,C 180,E1 29958.61,E2 29958.61} C_VEL
LIN {X 0,Y 114.146,Z 1203.685,A -85,B 0,C 180,E1 29981.31,E2 29981.31} C_VEL
LIN {X 0,Y 125.532,Z 1200.096,A -85,B 0,C 180,E1 30011.437,E2 30011.437} C_VEL
LIN {X 0,Y 140.276,Z 1194.818,A -85,B 0,C 180,E1 30024.492,E2 30024.492} C_VEL
LIN {X 0,Y 154.208,Z 1188.148,A -85,B 0,C 180,E1 30036.967,E2 30036.967} C_VEL
LIN {X 0,Y 217.314,Z 1159.961,A -85,B 0,C 180,E1 30053.317,E2 30053.317} C_VEL
LIN {X 0,Y 286.012,Z 1116.751,A -85,B 0,C 180,E1 30061.692,E2 30061.692} C_VEL
LIN {X 0,Y 303.544,Z 1102.99,A -85,B 0,C 180,E1 30063.168,E2 30063.168} C_VEL
LIN {X 0,Y 236.4,Z 1149.968,A -85,B 0,C 180,E1 30070.32,E2 30070.32} C_VEL
LIN {X 0,Y 169.213,Z 1183.488,A -85,B 0,C 180,E1 30084.161,E2 30084.161} C_VEL
LIN {X 0,Y 120.22,Z 1201.679,A -85,B 0,C 180,E1 30111.102,E2 30111.102} C_VEL
LIN {X 0,Y 106.844,Z 1206.042,A -85,B 0,C 180,E1 30146.129,E2 30146.129} C_VEL
LIN {X 0,Y 110.645,Z 1202.196,A -85,B 0,C 180,E1 30174.505,E2 30174.505} C_VEL
LIN {X 0,Y 142.502,Z 1185.906,A -85,B 0,C 180,E1 30205.873,E2 30205.873} C_VEL
LIN {X 0,Y 199.348,Z 1154.599,A -85,B 0,C 180,E1 30224.39,E2 30224.39} C_VEL
LIN {X 0,Y 260.187,Z 1110.605,A -85,B 0,C 180,E1 30233.717,E2 30233.717} C_VEL
LIN {X 0,Y 306.617,Z 1066.213,A -85,B 0,C 180,E1 30238.266,E2 30238.266} C_VEL
LIN {X 0,Y 307.89,Z 1063.289,A -85,B 0,C 180,E1 30244.275,E2 30244.275} C_VEL
LIN {X 0,Y 305.318,Z 1067.185,A -85,B 0,C 180,E1 30249.231,E2 30249.231} C_VEL
LIN {X 0,Y 246.235,Z 1121.12,A -85,B 0,C 180,E1 30255.353,E2 30255.353} C_VEL
LIN {X 0,Y 185.672,Z 1161.658,A -85,B 0,C 180,E1 30266.256,E2 30266.256} C_VEL
LIN {X 0,Y 133.833,Z 1188.545,A -85,B 0,C 180,E1 30286.925,E2 30286.925} C_VEL
LIN {X 0,Y 109.303,Z 1201.075,A -85,B 0,C 180,E1 30317.781,E2 30317.781} C_VEL
LIN {X 0,Y 106.121,Z 1203.786,A -85,B 0,C 180,E1 30342.177,E2 30342.177} C_VEL
LIN {X 0,Y 121.396,Z 1199.442,A -85,B 0,C 180,E1 30376.456,E2 30376.456} C_VEL
LIN {X 0,Y 154.208,Z 1188.148,A -85,B 0,C 180,E1 30396.967,E2 30396.967} C_VEL
LIN {X 0,Y 173.661,Z 1179.403,A -85,B 0,C 180,E1 30406.938,E2 30406.938} C_VEL
LIN {X 0,Y 240.544,Z 1146.539,A -85,B 0,C 180,E1 30418.815,E2 30418.815} C_VEL
LIN {X 0,Y 282.65,Z 1119.189,A -85,B 0,C 180,E1 30423.386,E2 30423.386} C_VEL
LIN {X 0,Y 215.967,Z 1160.593,A -85,B 0,C 180,E1 30430.937,E2 30430.937} C_VEL
LIN {X 0,Y 148.727,Z 1190.058,A -85,B 0,C 180,E1 30447.235,E2 30447.235} C_VEL
LIN {X 0,Y 105.132,Z 1204.242,A -85,B 0,C 180,E1 30479.896,E2 30479.896} C_VEL
LIN {X 0,Y 98.844,Z 1205.945,A -85,B 0,C 180,E1 30505.816,E2 30505.816} C_VEL
LIN {X 0,Y 103.257,Z 1202.054,A -85,B 0,C 180,E1 30536.388,E2 30536.388} C_VEL
LIN {X 0,Y 137.844,Z 1185.729,A -85,B 0,C 180,E1 30568.689,E2 30568.689} C_VEL
LIN {X 0,Y 197.235,Z 1154.255,A -85,B 0,C 180,E1 30586.763,E2 30586.763} C_VEL
LIN {X 0,Y 260.941,Z 1108.868,A -85,B 0,C 180,E1 30595.73,E2 30595.73} C_VEL
LIN {X 0,Y 301.493,Z 1070.756,A -85,B 0,C 180,E1 30599.596,E2 30599.596} C_VEL
LIN {X 0,Y 302.227,Z 1069.095,A -85,B 0,C 180,E1 30604.356,E2 30604.356} C_VEL
LIN {X 0,Y 299.233,Z 1072.864,A -85,B 0,C 180,E1 30608.109,E2 30608.109} C_VEL
LIN {X 0,Y 239.023,Z 1125.468,A -85,B 0,C 180,E1 30614.163,E2 30614.163} C_VEL
LIN {X 0,Y 176.689,Z 1165.043,A -85,B 0,C 180,E1 30625.341,E2 30625.341} C_VEL
LIN {X 0,Y 123.721,Z 1190.65,A -85,B 0,C 180,E1 30647.349,E2 30647.349} C_VEL
LIN {X 0,Y 101.473,Z 1201.221,A -85,B 0,C 180,E1 30676.822,E2 30676.822} C_VEL
LIN {X 0,Y 98.138,Z 1203.888,A -85,B 0,C 180,E1 30703.185,E2 30703.185} C_VEL
LIN {X 0,Y 115.637,Z 1199.449,A -85,B 0,C 180,E1 30739.547,E2 30739.547} C_VEL
LIN {X 0,Y 170.226,Z 1180.831,A -85,B 0,C 180,E1 30766.028,E2 30766.028} C_VEL
LIN {X 0,Y 173.661,Z 1179.403,A -85,B 0,C 180,E1 30766.938,E2 30766.938} C_VEL
LIN {X 0,Y 196.186,Z 1169.065,A -85,B 0,C 180,E1 30774.839,E2 30774.839} C_VEL
LIN {X 0,Y 262.758,Z 1132.796,A -85,B 0,C 180,E1 30783.325,E2 30783.325} C_VEL
LIN {X 0,Y 193.534,Z 1170.76,A -85,B 0,C 180,E1 30792.028,E2 30792.028} C_VEL
LIN {X 0,Y 131.041,Z 1194.739,A -85,B 0,C 180,E1 30810.056,E2 30810.056} C_VEL
LIN {X 0,Y 93.832,Z 1205.248,A -85,B 0,C 180,E1 30846.405,E2 30846.405} C_VEL
LIN {X 0,Y 90.815,Z 1205.446,A -85,B 0,C 180,E1 30875.029,E2 30875.029} C_VEL
LIN {X 0,Y 107.179,Z 1196.831,A -85,B 0,C 180,E1 30914.163,E2 30914.163} C_VEL
LIN {X 0,Y 159.322,Z 1173.567,A -85,B 0,C 180,E1 30940.862,E2 30940.862} C_VEL
LIN {X 0,Y 224.277,Z 1135.573,A -85,B 0,C 180,E1 30953.524,E2 30953.524} C_VEL
LIN {X 0,Y 287.75,Z 1084.023,A -85,B 0,C 180,E1 30959.936,E2 30959.936} C_VEL
LIN {X 0,Y 296.259,Z 1075.687,A -85,B 0,C 180,E1 30960.614,E2 30960.614} C_VEL
LIN {X 0,Y 295.67,Z 1075.99,A -85,B 0,C 180,E1 30966.433,E2 30966.433} C_VEL
LIN {X 0,Y 235.422,Z 1127.204,A -85,B 0,C 180,E1 30972.478,E2 30972.478} C_VEL
LIN {X 0,Y 170.005,Z 1167.195,A -85,B 0,C 180,E1 30983.747,E2 30983.747} C_VEL
LIN {X 0,Y 115.369,Z 1191.951,A -85,B 0,C 180,E1 31006.461,E2 31006.461} C_VEL
LIN {X 0,Y 91.65,Z 1202.712,A -85,B 0,C 180,E1 31045.017,E2 31045.017} C_VEL
LIN {X 0,Y 91.756,Z 1203.764,A -85,B 0,C 180,E1 31074.293,E2 31074.293} C_VEL
LIN {X 0,Y 120.061,Z 1196.854,A -85,B 0,C 180,E1 31110.148,E2 31110.148} C_VEL
LIN {X 0,Y 183.505,Z 1174.624,A -85,B 0,C 180,E1 31132.42,E2 31132.42} C_VEL
LIN {X 0,Y 196.186,Z 1169.065,A -85,B 0,C 180,E1 31134.839,E2 31134.839} C_VEL
LIN {X 0,Y 221.297,Z 1156.65,A -85,B 0,C 180,E1 31140.832,E2 31140.832} C_VEL
LIN {X 0,Y 241.352,Z 1145.825,A -85,B 0,C 180,E1 31143.423,E2 31143.423} C_VEL
LIN {X 0,Y 170.574,Z 1179.76,A -85,B 0,C 180,E1 31153.574,E2 31153.574} C_VEL
LIN {X 0,Y 106.443,Z 1200.415,A -85,B 0,C 180,E1 31178.696,E2 31178.696} C_VEL
LIN {X 0,Y 83.644,Z 1205.694,A -85,B 0,C 180,E1 31214.477,E2 31214.477} C_VEL
LIN {X 0,Y 82.804,Z 1205.327,A -85,B 0,C 180,E1 31235.517,E2 31235.517} C_VEL
LIN {X 0,Y 98.226,Z 1197.92,A -85,B 0,C 180,E1 31274.34,E2 31274.34} C_VEL
LIN {X 0,Y 151.646,Z 1175.779,A -85,B 0,C 180,E1 31302.359,E2 31302.359} C_VEL
LIN {X 0,Y 217.808,Z 1139.008,A -85,B 0,C 180,E1 31314.943,E2 31314.943} C_VEL
LIN {X 0,Y 281.122,Z 1089.819,A -85,B 0,C 180,E1 31321.113,E2 31321.113} C_VEL
LIN {X 0,Y 290.888,Z 1080.57,A -85,B 0,C 180,E1 31322.15,E2 31322.15} C_VEL
LIN {X 0,Y 290.346,Z 1080.964,A -85,B 0,C 180,E1 31325.285,E2 31325.285} C_VEL
LIN {X 0,Y 228.476,Z 1131.32,A -85,B 0,C 180,E1 31331.14,E2 31331.14} C_VEL
LIN {X 0,Y 161.592,Z 1170.025,A -85,B 0,C 180,E1 31342.458,E2 31342.458} C_VEL
LIN {X 0,Y 103.306,Z 1194.472,A -85,B 0,C 180,E1 31368.353,E2 31368.353} C_VEL
LIN {X 0,Y 83.662,Z 1202.834,A -85,B 0,C 180,E1 31404.54,E2 31404.54} C_VEL
LIN {X 0,Y 84.214,Z 1203.847,A -85,B 0,C 180,E1 31436.486,E2 31436.486} C_VEL
LIN {X 0,Y 117.181,Z 1196.482,A -85,B 0,C 180,E1 31474.583,E2 31474.583} C_VEL
LIN {X 0,Y 182.555,Z 1174.502,A -85,B 0,C 180,E1 31495.151,E2 31495.151} C_VEL
LIN {X 0,Y 221.297,Z 1156.65,A -85,B 0,C 180,E1 31500.832,E2 31500.832} C_VEL
LIN {X 0,Y 217.059,Z 1158.839,A -85,B 0,C 180,E1 31503.19,E2 31503.19} C_VEL
LIN {X 0,Y 195.252,Z 1169.086,A -85,B 0,C 180,E1 31506.481,E2 31506.481} C_VEL
LIN {X 0,Y 123.518,Z 1194.755,A -85,B 0,C 180,E1 31523.328,E2 31523.328} C_VEL
LIN {X 0,Y 79.128,Z 1205.133,A -85,B 0,C 180,E1 31561.664,E2 31561.664} C_VEL
LIN {X 0,Y 74.782,Z 1205.208,A -85,B 0,C 180,E1 31596.111,E2 31596.111} C_VEL
LIN {X 0,Y 92.468,Z 1197.73,A -85,B 0,C 180,E1 31637.939,E2 31637.939} C_VEL
LIN {X 0,Y 149.295,Z 1175.489,A -85,B 0,C 180,E1 31665.462,E2 31665.462} C_VEL
LIN {X 0,Y 216.856,Z 1138.838,A -85,B 0,C 180,E1 31677.137,E2 31677.137} C_VEL
LIN {X 0,Y 281.411,Z 1089.265,A -85,B 0,C 180,E1 31682.824,E2 31682.824} C_VEL
LIN {X 0,Y 284.89,Z 1085.985,A -85,B 0,C 180,E1 31683.61,E2 31683.61} C_VEL
LIN {X 0,Y 280.559,Z 1089.992,A -85,B 0,C 180,E1 31684.573,E2 31684.573} C_VEL
LIN {X 0,Y 215.475,Z 1139.339,A -85,B 0,C 180,E1 31690.408,E2 31690.408} C_VEL
LIN {X 0,Y 148.007,Z 1175.239,A -85,B 0,C 180,E1 31702.309,E2 31702.309} C_VEL
LIN {X 0,Y 93.091,Z 1196.198,A -85,B 0,C 180,E1 31729.007,E2 31729.007} C_VEL
LIN {X 0,Y 75.67,Z 1202.957,A -85,B 0,C 180,E1 31763.961,E2 31763.961} C_VEL
LIN {X 0,Y 76.837,Z 1203.926,A -85,B 0,C 180,E1 31799.262,E2 31799.262} C_VEL
LIN {X 0,Y 113.723,Z 1196.465,A -85,B 0,C 180,E1 31838.535,E2 31838.535} C_VEL
LIN {X 0,Y 184.095,Z 1173.511,A -85,B 0,C 180,E1 31858.263,E2 31858.263} C_VEL
LIN {X 0,Y 222.356,Z 1156.081,A -85,B 0,C 180,E1 31863.168,E2 31863.168} C_VEL
LIN {X 0,Y 195.252,Z 1169.086,A -85,B 0,C 180,E1 31866.481,E2 31866.481} C_VEL
LIN {X 0,Y 162.84,Z 1181.643,A -85,B 0,C 180,E1 31868.823,E2 31868.823} C_VEL
LIN {X 0,Y 96.918,Z 1200.385,A -85,B 0,C 180,E1 31890.999,E2 31890.999} C_VEL
LIN {X 0,Y 68.111,Z 1205.538,A -85,B 0,C 180,E1 31930.813,E2 31930.813} C_VEL
LIN {X 0,Y 66.788,Z 1205.088,A -85,B 0,C 180,E1 31956.845,E2 31956.845} C_VEL
LIN {X 0,Y 88.787,Z 1196.975,A -85,B 0,C 180,E1 32003.435,E2 32003.435} C_VEL
LIN {X 0,Y 150.842,Z 1173.609,A -85,B 0,C 180,E1 32029.483,E2 32029.483} C_VEL
LIN {X 0,Y 220.38,Z 1135.951,A -85,B 0,C 180,E1 32039.762,E2 32039.762} C_VEL
LIN {X 0,Y 266.489,Z 1102.096,A -85,B 0,C 180,E1 32043.821,E2 32043.821} C_VEL
LIN {X 0,Y 198.754,Z 1148.885,A -85,B 0,C 180,E1 32050.019,E2 32050.019} C_VEL
LIN {X 0,Y 128.827,Z 1182.081,A -85,B 0,C 180,E1 32063.699,E2 32063.699} C_VEL
LIN {X 0,Y 79.028,Z 1198.903,A -85,B 0,C 180,E1 32094.5,E2 32094.5} C_VEL
LIN {X 0,Y 67.698,Z 1203.079,A -85,B 0,C 180,E1 32123.247,E2 32123.247} C_VEL
LIN {X 0,Y 69.653,Z 1204.006,A -85,B 0,C 180,E1 32162.63,E2 32162.63} C_VEL
LIN {X 0,Y 110.636,Z 1196.499,A -85,B 0,C 180,E1 32202.631,E2 32202.631} C_VEL
LIN {X 0,Y 179.605,Z 1175.206,A -85,B 0,C 180,E1 32220.328,E2 32220.328} C_VEL
LIN {X 0,Y 201.047,Z 1166.271,A -85,B 0,C 180,E1 32223.256,E2 32223.256} C_VEL
LIN {X 0,Y 162.84,Z 1181.643,A -85,B 0,C 180,E1 32228.823,E2 32228.823} C_VEL
LIN {X 0,Y 129.933,Z 1191.58,A -85,B 0,C 180,E1 32232.43,E2 32232.43} C_VEL
LIN {X 0,Y 72.533,Z 1203.952,A -85,B 0,C 180,E1 32263.365,E2 32263.365} C_VEL
LIN {X 0,Y 58.757,Z 1205.452,A -85,B 0,C 180,E1 32302.949,E2 32302.949} C_VEL
LIN {X 0,Y 66.036,Z 1202.082,A -85,B 0,C 180,E1 32346.776,E2 32346.776} C_VEL
LIN {X 0,Y 118.258,Z 1185.656,A -85,B 0,C 180,E1 32384.889,E2 32384.889} C_VEL
LIN {X 0,Y 190.069,Z 1153.555,A -85,B 0,C 180,E1 32398.876,E2 32398.876} C_VEL
LIN {X 0,Y 240.965,Z 1121.693,A -85,B 0,C 180,E1 32403.624,E2 32403.624} C_VEL
LIN {X 0,Y 170.522,Z 1163.246,A -85,B 0,C 180,E1 32411.201,E2 32411.201} C_VEL
LIN {X 0,Y 103.73,Z 1189.858,A -85,B 0,C 180,E1 32428.209,E2 32428.209} C_VEL
LIN {X 0,Y 63.09,Z 1201.949,A -85,B 0,C 180,E1 32468.49,E2 32468.49} C_VEL
LIN {X 0,Y 58.799,Z 1204.392,A -85,B 0,C 180,E1 32512.377,E2 32512.377} C_VEL
LIN {X 0,Y 89.74,Z 1200.274,A -85,B 0,C 180,E1 32557.78,E2 32557.78} C_VEL
LIN {X 0,Y 161.396,Z 1181.718,A -85,B 0,C 180,E1 32580.376,E2 32580.376} C_VEL
LIN {X 0,Y 179.659,Z 1175.17,A -85,B 0,C 180,E1 32583.102,E2 32583.102} C_VEL
LIN {X 0,Y 129.933,Z 1191.58,A -85,B 0,C 180,E1 32592.43,E2 32592.43} C_VEL
LIN {X 0,Y 97.147,Z 1198.885,A -85,B 0,C 180,E1 32598.291,E2 32598.291} C_VEL
LIN {X 0,Y 53.028,Z 1205.381,A -85,B 0,C 180,E1 32645.03,E2 32645.03} C_VEL
LIN {X 0,Y 50.8,Z 1204.848,A -85,B 0,C 180,E1 32679.015,E2 32679.015} C_VEL
LIN {X 0,Y 78.009,Z 1197.161,A -85,B 0,C 180,E1 32731.647,E2 32731.647} C_VEL
LIN {X 0,Y 145.015,Z 1174.6,A -85,B 0,C 180,E1 32755.241,E2 32755.241} C_VEL
LIN {X 0,Y 214.656,Z 1139.141,A -85,B 0,C 180,E1 32763.769,E2 32763.769} C_VEL
LIN {X 0,Y 144.04,Z 1174.638,A -85,B 0,C 180,E1 32772.458,E2 32772.458} C_VEL
LIN {X 0,Y 75.142,Z 1197.165,A -85,B 0,C 180,E1 32798.107,E2 32798.107} C_VEL
LIN {X 0,Y 51.757,Z 1203.324,A -85,B 0,C 180,E1 32841.153,E2 32841.153} C_VEL
LIN {X 0,Y 56.249,Z 1204.165,A -85,B 0,C 180,E1 32891.89,E2 32891.89} C_VEL
LIN {X 0,Y 109.471,Z 1195.856,A -85,B 0,C 180,E1 32932.532,E2 32932.532} C_VEL
LIN {X 0,Y 159.187,Z 1182.501,A -85,B 0,C 180,E1 32943.195,E2 32943.195} C_VEL
LIN {X 0,Y 97.147,Z 1198.885,A -85,B 0,C 180,E1 32958.291,E2 32958.291} C_VEL
LIN {X 0,Y 65.468,Z 1203.407,A -85,B 0,C 180,E1 32969.425,E2 32969.425} C_VEL
LIN {X 0,Y 42.792,Z 1205.254,A -85,B 0,C 180,E1 33020.297,E2 33020.297} C_VEL
LIN {X 0,Y 53.097,Z 1201.939,A -85,B 0,C 180,E1 33076.172,E2 33076.172} C_VEL
LIN {X 0,Y 115.03,Z 1185.171,A -85,B 0,C 180,E1 33112.985,E2 33112.985} C_VEL
LIN {X 0,Y 185.703,Z 1155.332,A -85,B 0,C 180,E1 33123.531,E2 33123.531} C_VEL
LIN {X 0,Y 117.594,Z 1183.938,A -85,B 0,C 180,E1 33133.862,E2 33133.862} C_VEL
LIN {X 0,Y 56.191,Z 1200.554,A -85,B 0,C 180,E1 33167.023,E2 33167.023} C_VEL
LIN {X 0,Y 43.813,Z 1203.446,A -85,B 0,C 180,E1 33199.532,E2 33199.532} C_VEL
LIN {X 0,Y 50.314,Z 1204.246,A -85,B 0,C 180,E1 33258.285,E2 33258.285} C_VEL
LIN {X 0,Y 113.472,Z 1194.827,A -85,B 0,C 180,E1 33298.29,E2 33298.29} C_VEL
LIN {X 0,Y 137.877,Z 1188.915,A -85,B 0,C 180,E1 33303.07,E2 33303.07} C_VEL
LIN {X 0,Y 65.468,Z 1203.407,A -85,B 0,C 180,E1 33329.425,E2 33329.425} C_VEL
LIN {X 0,Y 38.488,Z 1205.221,A -85,B 0,C 180,E1 33355.979,E2 33355.979} C_VEL
LIN {X 0,Y 34.918,Z 1204.607,A -85,B 0,C 180,E1 33403.178,E2 33403.178} C_VEL
LIN {X 0,Y 71.608,Z 1196.774,A -85,B 0,C 180,E1 33463.477,E2 33463.477} C_VEL
LIN {X 0,Y 144.597,Z 1174.008,A -85,B 0,C 180,E1 33481.934,E2 33481.934} C_VEL
LIN {X 0,Y 159.802,Z 1167.709,A -85,B 0,C 180,E1 33483.751,E2 33483.751} C_VEL
LIN {X 0,Y 87.797,Z 1192.388,A -85,B 0,C 180,E1 33497.304,E2 33497.304} C_VEL
LIN {X 0,Y 41.63,Z 1202.383,A -85,B 0,C 180,E1 33536.242,E2 33536.242} C_VEL
LIN {X 0,Y 33.734,Z 1204.329,A -85,B 0,C 180,E1 33582.345,E2 33582.345} C_VEL
LIN {X 0,Y 69.362,Z 1202.136,A -85,B 0,C 180,E1 33648.229,E2 33648.229} C_VEL
LIN {X 0,Y 113.646,Z 1194.809,A -85,B 0,C 180,E1 33663.605,E2 33663.605} C_VEL
LIN {X 0,Y 47.254,Z 1204.836,A -85,B 0,C 180,E1 33697.363,E2 33697.363} C_VEL
LIN {X 0,Y 38.488,Z 1205.221,A -85,B 0,C 180,E1 33715.979,E2 33715.979} C_VEL
LIN {X 0,Y 28.44,Z 1204.092,A -85,B 0,C 180,E1 33778.414,E2 33778.414} C_VEL
LIN {X 0,Y 76.637,Z 1195.012,A -85,B 0,C 180,E1 33832.688,E2 33832.688} C_VEL
LIN {X 0,Y 129.659,Z 1179.466,A -85,B 0,C 180,E1 33844.004,E2 33844.004} C_VEL
LIN {X 0,Y 58.196,Z 1198.56,A -85,B 0,C 180,E1 33863.23,E2 33863.23} C_VEL
LIN {X 0,Y 28.112,Z 1203.69,A -85,B 0,C 180,E1 33913.551,E2 33913.551} C_VEL
LIN {X 0,Y 41.067,Z 1204.407,A -85,B 0,C 180,E1 33996.142,E2 33996.142} C_VEL
LIN {X 0,Y 90.902,Z 1199.078,A -85,B 0,C 180,E1 34022.558,E2 34022.558} C_VEL
LIN {X 0,Y 42.764,Z 1204.762,A -85,B 0,C 180,E1 34048.567,E2 34048.567} C_VEL
LIN {X 0,Y 27.099,Z 1204.485,A -85,B 0,C 180,E1 34127.083,E2 34127.083} C_VEL
LIN {X 0,Y 28.44,Z 1204.092,A -85,B 0,C 180,E1 34138.414,E2 34138.414} C_VEL
LIN {X 0,Y 46.717,Z 1200.489,A -85,B 0,C 180,E1 34187.389,E2 34187.389} C_VEL
LIN {X 0,Y 99.234,Z 1189.052,A -85,B 0,C 180,E1 34203.967,E2 34203.967} C_VEL
LIN {X 0,Y 29.645,Z 1202.671,A -85,B 0,C 180,E1 34238.708,E2 34238.708} C_VEL
LIN {X 0,Y 18.063,Z 1204.531,A -85,B 0,C 180,E1 34313.534,E2 34313.534} C_VEL
LIN {X 0,Y 67.973,Z 1202.204,A -85,B 0,C 180,E1 34382.605,E2 34382.605} C_VEL
LIN {X 0,Y 19.318,Z 1204.956,A -85,B 0,C 180,E1 34448.078,E2 34448.078} C_VEL
LIN {X 0,Y 40.161,Z 1201.502,A -85,B 0,C 180,E1 34542.516,E2 34542.516} C_VEL
LIN {X 0,Y 46.717,Z 1200.489,A -85,B 0,C 180,E1 34547.389,E2 34547.389} C_VEL
LIN {X 0,Y 64.999,Z 1196.97,A -85,B 0,C 180,E1 34563.142,E2 34563.142} C_VEL
LIN {X 0,Y 67.303,Z 1196.507,A -85,B 0,C 180,E1 34563.622,E2 34563.622} C_VEL
LIN {X 0,Y 13.406,Z 1203.934,A -85,B 0,C 180,E1 34613.573,E2 34613.573} C_VEL
LIN {X 0,Y 42.839,Z 1204.306,A -85,B 0,C 180,E1 34742.87,E2 34742.87} C_VEL
LIN {X 0,Y 12.183,Z 1204.856,A -85,B 0,C 180,E1 34793.7,E2 34793.7} C_VEL
LIN {X 0,Y 38.495,Z 1201.356,A -85,B 0,C 180,E1 34914.32,E2 34914.32} C_VEL
LIN {X 0,Y 64.999,Z 1196.97,A -85,B 0,C 180,E1 34923.142,E2 34923.142} C_VEL
LIN {X 0,Y 67.316,Z 1198.933,A -85,B 0,C 180,E1 34923.625,E2 34923.625} C_VEL
LIN {X 0,Y 67.316,Z 1212.987,A -85,B 0,C 180,E1 34923.625,E2 34923.625} C_VEL
LIN {X 0,Y 25.533,Z 1212.987,A -85,B 0,C 180,E1 34930.154,E2 34930.154} C_VEL
LIN {X 0,Y 23.569,Z 1210.987,A -85,B 0,C 180,E1 34931.04,E2 34931.04} C_VEL
LIN {X 0,Y 23.569,Z 1204.958,A -85,B 0,C 180,E1 34931.04,E2 34931.04} C_VEL
LIN {X 0,Y 23.265,Z 1202.958,A -85,B 0,C 180,E1 34926.113,E2 34926.113} C_VEL
LIN {X 0,Y 7.413,Z 1204.757,A -85,B 0,C 180,E1 34753.344,E2 34753.344} C_VEL
LIN {X 0,Y 8.403,Z 1204.056,A -85,B 0,C 180,E1 34578.686,E2 34578.686} C_VEL
LIN {X 0,Y 23.265,Z 1202.958,A -85,B 0,C 180,E1 34566.113,E2 34566.113} C_VEL
LIN {X 0,Y 25.395,Z 1204.953,A -85,B 0,C 180,E1 34565.53,E2 34565.53} C_VEL
LIN {X 0,Y 25.395,Z 1215,A -85,B 0,C 180,E1 34565.53,E2 34565.53} C_VEL
LIN {X 0,Y 25.395,Z 1215,A -85,B 0,C 180,E1 34565.53,E2 34565.53}

QRS_NEXT_CUT()
PTP {E1 34737.172,E2 34737.172}
PTP {X 0,Y 759.916,A -85,B 0,C 180,E1 34737.172,E2 34737.172,E3 0,E4 0,E5 0,E6 0}
QRS_SPEED_INIT()
LIN {X 0,Y 759.916,Z 1215,A -85,B 0,C 180,E1 34737.172,E2 34737.172,E3 0,E4 0,E5 0,E6 0} C_VEL
LIN {X 0,Y 759.916,Z 329.651,A -85,B 0,C 180,E1 34737.172,E2 34737.172} C_VEL
LIN {X 0,Y 759.916,Z 321.577,A -85,B 0,C 180,E1 34737.172,E2 34737.172} C_VEL
LIN {X 0,Y 759.916,Z 319.577,A -85,B 0,C 180,E1 34737.021,E2 34737.021} C_VEL
LIN {X 0,Y 759.849,Z 319.574,A -85,B 0,C 180,E1 34734.336,E2 34734.336} C_VEL
LIN {X 0,Y 759.851,Z 319.571,A -85,B 0,C 180,E1 34731.83,E2 34731.83} C_VEL
LIN {X 0,Y 759.913,Z 319.569,A -85,B 0,C 180,E1 34729.078,E2 34729.078} C_VEL
LIN {X 0,Y 759.858,Z 319.574,A -85,B 0,C 180,E1 34726.221,E2 34726.221} C_VEL
LIN {X 0,Y 759.848,Z 319.571,A -85,B 0,C 180,E1 34723.722,E2 34723.722} C_VEL
LIN {X 0,Y 759.909,Z 319.567,A -85,B 0,C 180,E1 34721.034,E2 34721.034} C_VEL
LIN {X 0,Y 759.867,Z 319.575,A -85,B 0,C 180,E1 34718.055,E2 34718.055} C_VEL
LIN {X 0,Y 759.848,Z 319.571,A -85,B 0,C 180,E1 34715.511,E2 34715.511} C_VEL
LIN {X 0,Y 759.909,Z 319.567,A -85,B 0,C 180,E1 34712.804,E2 34712.804} C_VEL
LIN {X 0,Y 759.87,Z 319.575,A -85,B 0,C 180,E1 34709.823,E2 34709.823} C_VEL
LIN {X 0,Y 759.851,Z 319.572,A -85,B 0,C 180,E1 34707.259,E2 34707.259} C_VEL
LIN {X 0,Y 759.902,Z 319.567,A -85,B 0,C 180,E1 34704.622,E2 34704.622} C_VEL
LIN {X 0,Y 759.874,Z 319.576,A -85,B 0,C 180,E1 34701.604,E2 34701.604} C_VEL
LIN {X 0,Y 759.856,Z 319.58,A -85,B 0,C 180,E1 34699.282,E2 34699.282} C_VEL
LIN {X 0,Y 759.914,Z 341.188,A -85,B 0,C 180,E1 34697.866,E2 34697.866} C_VEL
LIN {X 0,Y 759.913,Z 553.045,A -85,B 0,C 180,E1 34695.319,E2 34695.319} C_VEL
LIN {X 0,Y 759.913,Z 778.061,A -85,B 0,C 180,E1 34692.708,E2 34692.708} C_VEL
LIN {X 0,Y 759.914,Z 821.22,A -85,B 0,C 180,E1 34692.187,E2 34692.187} C_VEL
LIN {X 0,Y 759.906,Z 846.697,A -85,B 0,C 180,E1 34691.742,E2 34691.742} C_VEL
LIN {X 0,Y 759.916,Z 873.487,A -85,B 0,C 180,E1 34691.12,E2 34691.12} C_VEL
LIN {X 0,Y 759.908,Z 896.825,A -85,B 0,C 180,E1 34690.441,E2 34690.441} C_VEL
LIN {X 0,Y 759.918,Z 920.733,A -85,B 0,C 180,E1 34689.628,E2 34689.628} C_VEL
LIN {X 0,Y 759.917,Z 946.582,A -85,B 0,C 180,E1 34688.584,E2 34688.584} C_VEL
LIN {X 0,Y 759.91,Z 967.501,A -85,B 0,C 180,E1 34687.616,E2 34687.616} C_VEL
LIN {X 0,Y 759.911,Z 986.849,A -85,B 0,C 180,E1 34686.617,E2 34686.617} C_VEL
LIN {X 0,Y 759.904,Z 1007.745,A -85,B 0,C 180,E1 34685.419,E2 34685.419} C_VEL
LIN {X 0,Y 759.916,Z 1031.031,A -85,B 0,C 180,E1 34683.909,E2 34683.909} C_VEL
LIN {X 0,Y 759.917,Z 1049.182,A -85,B 0,C 180,E1 34682.597,E2 34682.597} C_VEL
LIN {X 0,Y 759.909,Z 1068.631,A -85,B 0,C 180,E1 34681.049,E2 34681.049} C_VEL
LIN {X 0,Y 759.912,Z 1087.064,A -85,B 0,C 180,E1 34679.392,E2 34679.392} C_VEL
LIN {X 0,Y 759.905,Z 1101.781,A -85,B 0,C 180,E1 34677.931,E2 34677.931} C_VEL
LIN {X 0,Y 759.912,Z 1117.239,A -85,B 0,C 180,E1 34676.237,E2 34676.237} C_VEL
LIN {X 0,Y 759.892,Z 1132.599,A -85,B 0,C 180,E1 34674.321,E2 34674.321} C_VEL
LIN {X 0,Y 759.91,Z 1143.935,A -85,B 0,C 180,E1 34672.723,E2 34672.723} C_VEL
LIN {X 0,Y 759.898,Z 1153.506,A -85,B 0,C 180,E1 34671.213,E2 34671.213} C_VEL
LIN {X 0,Y 759.917,Z 1162.101,A -85,B 0,C 180,E1 34669.684,E2 34669.684} C_VEL
LIN {X 0,Y 759.89,Z 1170.303,A -85,B 0,C 180,E1 34668.012,E2 34668.012} C_VEL
LIN {X 0,Y 759.913,Z 1178.18,A -85,B 0,C 180,E1 34666.118,E2 34666.118} C_VEL
LIN {X 0,Y 759.918,Z 1184.829,A -85,B 0,C 180,E1 34664.088,E2 34664.088} C_VEL
LIN {X 0,Y 759.915,Z 1189.769,A -85,B 0,C 180,E1 34662.076,E2 34662.076} C_VEL
LIN {X 0,Y 759.912,Z 1193.155,A -85,B 0,C 180,E1 34660.002,E2 34660.002} C_VEL
LIN {X 0,Y 759.906,Z 1194.668,A -85,B 0,C 180,E1 34658.093,E2 34658.093} C_VEL
LIN {X 0,Y 759.908,Z 1194.825,A -85,B 0,C 180,E1 34656.346,E2 34656.346} C_VEL
LIN {X 0,Y 759.905,Z 1193.813,A -85,B 0,C 180,E1 34654.528,E2 34654.528} C_VEL
LIN {X 0,Y 759.908,Z 1190.902,A -85,B 0,C 180,E1 34652.413,E2 34652.413} C_VEL
LIN {X 0,Y 759.912,Z 1186.164,A -85,B 0,C 180,E1 34650.302,E2 34650.302} C_VEL
LIN {X 0,Y 759.917,Z 1180.138,A -85,B 0,C 180,E1 34648.341,E2 34648.341} C_VEL
LIN {X 0,Y 759.888,Z 1172.524,A -85,B 0,C 180,E1 34646.379,E2 34646.379} C_VEL
LIN {X 0,Y 759.896,Z 1163.092,A -85,B 0,C 180,E1 34644.412,E2 34644.412} C_VEL
LIN {X 0,Y 759.913,Z 1154.124,A -85,B 0,C 180,E1 34642.8,E2 34642.8} C_VEL
LIN {X 0,Y 759.893,Z 1144.671,A -85,B 0,C 180,E1 34641.297,E2 34641.297} C_VEL
LIN {X 0,Y 759.917,Z 1133.915,A -85,B 0,C 180,E1 34639.769,E2 34639.769} C_VEL
LIN {X 0,Y 759.889,Z 1121.271,A -85,B 0,C 180,E1 34638.155,E2 34638.155} C_VEL
LIN {X 0,Y 759.892,Z 1103.821,A -85,B 0,C 180,E1 34636.189,E2 34636.189} C_VEL
LIN {X 0,Y 759.91,Z 1088.596,A -85,B 0,C 180,E1 34634.665,E2 34634.665} C_VEL
LIN {X 0,Y 759.901,Z 1072.22,A -85,B 0,C 180,E1 34633.174,E2 34633.174} C_VEL
LIN {X 0,Y 759.915,Z 1051.298,A -85,B 0,C 180,E1 34631.473,E2 34631.473} C_VEL
LIN {X 0,Y 759.899,Z 1033.251,A -85,B 0,C 180,E1 34630.155,E2 34630.155} C_VEL
LIN {X 0,Y 759.912,Z 1013.205,A -85,B 0,C 180,E1 34628.828,E2 34628.828} C_VEL
LIN {X 0,Y 759.913,Z 989.552,A -85,B 0,C 180,E1 34627.439,E2 34627.439} C_VEL
LIN {X 0,Y 759.914,Z 969.28,A -85,B 0,C 180,E1 34626.382,E2 34626.382} C_VEL
LIN {X 0,Y 759.913,Z 949.893,A -85,B 0,C 180,E1 34625.473,E2 34625.473} C_VEL
LIN {X 0,Y 759.92,Z 929.99,A -85,B 0,C 180,E1 34624.641,E2 34624.641} C_VEL
LIN {X 0,Y 759.917,Z 908.416,A -85,B 0,C 180,E1 34623.847,E2 34623.847} C_VEL
LIN {X 0,Y 759.908,Z 879.321,A -85,B 0,C 180,E1 34622.947,E2 34622.947} C_VEL
LIN {X 0,Y 759.917,Z 853.746,A -85,B 0,C 180,E1 34622.317,E2 34622.317} C_VEL
LIN {X 0,Y 759.916,Z 827.086,A -85,B 0,C 180,E1 34621.813,E2 34621.813} C_VEL
LIN {X 0,Y 759.908,Z 799.731,A -85,B 0,C 180,E1 34621.448,E2 34621.448} C_VEL
LIN {X 0,Y 759.907,Z 578.437,A -85,B 0,C 180,E1 34618.89,E2 34618.89} C_VEL
LIN {X 0,Y 759.891,Z 367.287,A -85,B 0,C 180,E1 34616.362,E2 34616.362} C_VEL
LIN {X 0,Y 759.91,Z 340.577,A -85,B 0,C 180,E1 34616.023,E2 34616.023} C_VEL
LIN {X 0,Y 759.824,Z 319.583,A -85,B 0,C 180,E1 34614.62,E2 34614.62} C_VEL
LIN {X 0,Y 759.871,Z 319.577,A -85,B 0,C 180,E1 34611.702,E2 34611.702} C_VEL
LIN {X 0,Y 759.813,Z 319.577,A -85,B 0,C 180,E1 34609.155,E2 34609.155} C_VEL
LIN {X 0,Y 759.806,Z 319.577,A -85,B 0,C 180,E1 34606.918,E2 34606.918} C_VEL
LIN {X 0,Y 759.805,Z 319.577,A -85,B 0,C 180,E1 34604.753,E2 34604.753} C_VEL
LIN {X 0,Y 759.809,Z 319.576,A -85,B 0,C 180,E1 34602.564,E2 34602.564} C_VEL
LIN {X 0,Y 759.827,Z 319.577,A -85,B 0,C 180,E1 34600.251,E2 34600.251} C_VEL
LIN {X 0,Y 759.879,Z 319.575,A -85,B 0,C 180,E1 34597.345,E2 34597.345} C_VEL
LIN {X 0,Y 759.819,Z 319.576,A -85,B 0,C 180,E1 34594.802,E2 34594.802} C_VEL
LIN {X 0,Y 759.81,Z 319.576,A -85,B 0,C 180,E1 34592.564,E2 34592.564} C_VEL
LIN {X 0,Y 759.81,Z 319.576,A -85,B 0,C 180,E1 34590.354,E2 34590.354} C_VEL
LIN {X 0,Y 759.814,Z 319.575,A -85,B 0,C 180,E1 34588.156,E2 34588.156} C_VEL
LIN {X 0,Y 759.846,Z 319.576,A -85,B 0,C 180,E1 34585.738,E2 34585.738} C_VEL
LIN {X 0,Y 759.841,Z 319.574,A -85,B 0,C 180,E1 34582.679,E2 34582.679} C_VEL
LIN {X 0,Y 759.817,Z 319.575,A -85,B 0,C 180,E1 34580.329,E2 34580.329} C_VEL
LIN {X 0,Y 759.813,Z 319.576,A -85,B 0,C 180,E1 34578.094,E2 34578.094} C_VEL
LIN {X 0,Y 759.817,Z 319.576,A -85,B 0,C 180,E1 34575.86,E2 34575.86} C_VEL
LIN {X 0,Y 759.852,Z 319.577,A -85,B 0,C 180,E1 34573.391,E2 34573.391} C_VEL
LIN {X 0,Y 759.849,Z 319.574,A -85,B 0,C 180,E1 34570.386,E2 34570.386} C_VEL
LIN {X 0,Y 759.818,Z 319.575,A -85,B 0,C 180,E1 34567.942,E2 34567.942} C_VEL
LIN {X 0,Y 759.817,Z 319.575,A -85,B 0,C 180,E1 34565.74,E2 34565.74} C_VEL
LIN {X 0,Y 759.823,Z 319.576,A -85,B 0,C 180,E1 34563.47,E2 34563.47} C_VEL
LIN {X 0,Y 759.892,Z 319.577,A -85,B 0,C 180,E1 34560.829,E2 34560.829} C_VEL
LIN {X 0,Y 759.841,Z 319.574,A -85,B 0,C 180,E1 34557.964,E2 34557.964} C_VEL
LIN {X 0,Y 759.822,Z 319.574,A -85,B 0,C 180,E1 34555.623,E2 34555.623} C_VEL
LIN {X 0,Y 759.82,Z 319.575,A -85,B 0,C 180,E1 34553.35,E2 34553.35} C_VEL
LIN {X 0,Y 759.836,Z 319.576,A -85,B 0,C 180,E1 34550.991,E2 34550.991} C_VEL
LIN {X 0,Y 759.912,Z 319.571,A -85,B 0,C 180,E1 34548.155,E2 34548.155} C_VEL
LIN {X 0,Y 759.829,Z 319.574,A -85,B 0,C 180,E1 34545.443,E2 34545.443} C_VEL
LIN {X 0,Y 759.823,Z 319.575,A -85,B 0,C 180,E1 34543.093,E2 34543.093} C_VEL
LIN {X 0,Y 759.839,Z 319.575,A -85,B 0,C 180,E1 34540.713,E2 34540.713} C_VEL
LIN {X 0,Y 759.905,Z 319.572,A -85,B 0,C 180,E1 34537.812,E2 34537.812} C_VEL
LIN {X 0,Y 759.832,Z 319.572,A -85,B 0,C 180,E1 34535.179,E2 34535.179} C_VEL
LIN {X 0,Y 759.826,Z 319.575,A -85,B 0,C 180,E1 34532.817,E2 34532.817} C_VEL
LIN {X 0,Y 759.842,Z 319.576,A -85,B 0,C 180,E1 34530.431,E2 34530.431} C_VEL
LIN {X 0,Y 759.9,Z 319.571,A -85,B 0,C 180,E1 34527.502,E2 34527.502} C_VEL
LIN {X 0,Y 759.834,Z 319.573,A -85,B 0,C 180,E1 34524.896,E2 34524.896} C_VEL
LIN {X 0,Y 759.828,Z 319.574,A -85,B 0,C 180,E1 34522.557,E2 34522.557} C_VEL
LIN {X 0,Y 759.845,Z 319.576,A -85,B 0,C 180,E1 34520.145,E2 34520.145} C_VEL
LIN {X 0,Y 759.903,Z 319.572,A -85,B 0,C 180,E1 34517.237,E2 34517.237} C_VEL
LIN {X 0,Y 759.836,Z 319.574,A -85,B 0,C 180,E1 34514.609,E2 34514.609} C_VEL
LIN {X 0,Y 759.875,Z 319.645,A -85,B 0,C 180,E1 34512.942,E2 34512.942} C_VEL
LIN {X 0,Y 759.894,Z 350.99,A -85,B 0,C 180,E1 34510.914,E2 34510.914} C_VEL
LIN {X 0,Y 759.916,Z 561.522,A -85,B 0,C 180,E1 34508.381,E2 34508.381} C_VEL
LIN {X 0,Y 759.919,Z 788.685,A -85,B 0,C 180,E1 34505.746,E2 34505.746} C_VEL
LIN {X 0,Y 759.911,Z 830.473,A -85,B 0,C 180,E1 34505.243,E2 34505.243} C_VEL
LIN {X 0,Y 759.909,Z 856.604,A -85,B 0,C 180,E1 34504.789,E2 34504.789} C_VEL
LIN {X 0,Y 759.913,Z 883.606,A -85,B 0,C 180,E1 34504.163,E2 34504.163} C_VEL
LIN {X 0,Y 759.907,Z 907.507,A -85,B 0,C 180,E1 34503.465,E2 34503.465} C_VEL
LIN {X 0,Y 759.918,Z 931.763,A -85,B 0,C 180,E1 34502.637,E2 34502.637} C_VEL
LIN {X 0,Y 759.917,Z 956.967,A -85,B 0,C 180,E1 34501.611,E2 34501.611} C_VEL
LIN {X 0,Y 759.912,Z 976.745,A -85,B 0,C 180,E1 34500.698,E2 34500.698} C_VEL
LIN {X 0,Y 759.913,Z 995.427,A -85,B 0,C 180,E1 34499.738,E2 34499.738} C_VEL
LIN {X 0,Y 759.909,Z 1013.707,A -85,B 0,C 180,E1 34498.702,E2 34498.702} C_VEL
LIN {X 0,Y 759.911,Z 1035.516,A -85,B 0,C 180,E1 34497.335,E2 34497.335} C_VEL
LIN {X 0,Y 759.912,Z 1056.845,A -85,B 0,C 180,E1 34495.818,E2 34495.818} C_VEL
LIN {X 0,Y 759.91,Z 1073.823,A -85,B 0,C 180,E1 34494.485,E2 34494.485} C_VEL
LIN {X 0,Y 759.901,Z 1092.853,A -85,B 0,C 180,E1 34492.84,E2 34492.84} C_VEL
LIN {X 0,Y 759.895,Z 1109.495,A -85,B 0,C 180,E1 34491.213,E2 34491.213} C_VEL
LIN {X 0,Y 759.905,Z 1122.958,A -85,B 0,C 180,E1 34489.764,E2 34489.764} C_VEL
LIN {X 0,Y 759.897,Z 1135.732,A -85,B 0,C 180,E1 34488.249,E2 34488.249} C_VEL
LIN {X 0,Y 759.909,Z 1150.031,A -85,B 0,C 180,E1 34486.354,E2 34486.354} C_VEL
LIN {X 0,Y 759.909,Z 1162.194,A -85,B 0,C 180,E1 34484.477,E2 34484.477} C_VEL
LIN {X 0,Y 759.91,Z 1171.058,A -85,B 0,C 180,E1 34482.925,E2 34482.925} C_VEL
LIN {X 0,Y 759.91,Z 1178.784,A -85,B 0,C 180,E1 34481.383,E2 34481.383} C_VEL
LIN {X 0,Y 759.906,Z 1186.43,A -85,B 0,C 180,E1 34479.619,E2 34479.619} C_VEL
LIN {X 0,Y 759.908,Z 1193.594,A -85,B 0,C 180,E1 34477.561,E2 34477.561} C_VEL
LIN {X 0,Y 759.91,Z 1199.108,A -85,B 0,C 180,E1 34475.436,E2 34475.436} C_VEL
LIN {X 0,Y 759.916,Z 1202.585,A -85,B 0,C 180,E1 34473.47,E2 34473.47} C_VEL
LIN {X 0,Y 759.914,Z 1204.58,A -85,B 0,C 180,E1 34471.432,E2 34471.432} C_VEL
LIN {X 0,Y 759.889,Z 1204.849,A -85,B 0,C 180,E1 34469.472,E2 34469.472} C_VEL
LIN {X 0,Y 759.907,Z 1203.907,A -85,B 0,C 180,E1 34467.662,E2 34467.662} C_VEL
LIN {X 0,Y 759.908,Z 1201.054,A -85,B 0,C 180,E1 34465.548,E2 34465.548} C_VEL
LIN {X 0,Y 759.914,Z 1196.566,A -85,B 0,C 180,E1 34463.503,E2 34463.503} C_VEL
LIN {X 0,Y 759.912,Z 1190.629,A -85,B 0,C 180,E1 34461.526,E2 34461.526} C_VEL
LIN {X 0,Y 759.896,Z 1182.68,A -85,B 0,C 180,E1 34459.462,E2 34459.462} C_VEL
LIN {X 0,Y 759.905,Z 1173.111,A -85,B 0,C 180,E1 34457.461,E2 34457.461} C_VEL
LIN {X 0,Y 759.91,Z 1164.056,A -85,B 0,C 180,E1 34455.834,E2 34455.834} C_VEL
LIN {X 0,Y 759.894,Z 1154.212,A -85,B 0,C 180,E1 34454.273,E2 34454.273} C_VEL
LIN {X 0,Y 759.904,Z 1143.666,A -85,B 0,C 180,E1 34452.78,E2 34452.78} C_VEL
LIN {X 0,Y 759.896,Z 1130.456,A -85,B 0,C 180,E1 34451.1,E2 34451.1} C_VEL
LIN {X 0,Y 759.898,Z 1113.394,A -85,B 0,C 180,E1 34449.191,E2 34449.191} C_VEL
LIN {X 0,Y 759.898,Z 1098.828,A -85,B 0,C 180,E1 34447.732,E2 34447.732} C_VEL
LIN {X 0,Y 759.911,Z 1082.654,A -85,B 0,C 180,E1 34446.258,E2 34446.258} C_VEL
LIN {X 0,Y 759.91,Z 1061.274,A -85,B 0,C 180,E1 34444.516,E2 34444.516} C_VEL
LIN {X 0,Y 759.91,Z 1044.049,A -85,B 0,C 180,E1 34443.257,E2 34443.257} C_VEL
LIN {X 0,Y 759.914,Z 1026.242,A -85,B 0,C 180,E1 34442.069,E2 34442.069} C_VEL
LIN {X 0,Y 759.905,Z 1003.453,A -85,B 0,C 180,E1 34440.695,E2 34440.695} C_VEL
LIN {X 0,Y 759.916,Z 981.266,A -85,B 0,C 180,E1 34439.525,E2 34439.525} C_VEL
LIN {X 0,Y 759.912,Z 961.681,A -85,B 0,C 180,E1 34438.598,E2 34438.598} C_VEL
LIN {X 0,Y 759.918,Z 942.461,A -85,B 0,C 180,E1 34437.785,E2 34437.785} C_VEL
LIN {X 0,Y 759.919,Z 923.853,A -85,B 0,C 180,E1 34437.085,E2 34437.085} C_VEL
LIN {X 0,Y 759.909,Z 905.51,A -85,B 0,C 180,E1 34436.474,E2 34436.474} C_VEL
LIN {X 0,Y 759.913,Z 882.834,A -85,B 0,C 180,E1 34435.818,E2 34435.818} C_VEL
LIN {X 0,Y 759.911,Z 855.67,A -85,B 0,C 180,E1 34435.191,E2 34435.191} C_VEL
LIN {X 0,Y 759.91,Z 829.101,A -85,B 0,C 180,E1 34434.737,E2 34434.737} C_VEL
LIN {X 0,Y 759.915,Z 735.994,A -85,B 0,C 180,E1 34433.651,E2 34433.651} C_VEL
LIN {X 0,Y 759.912,Z 513.174,A -85,B 0,C 180,E1 34431.045,E2 34431.045} C_VEL
LIN {X 0,Y 759.895,Z 350.57,A -85,B 0,C 180,E1 34429.073,E2 34429.073} C_VEL
LIN {X 0,Y 759.879,Z 319.576,A -85,B 0,C 180,E1 34427.032,E2 34427.032} C_VEL
LIN {X 0,Y 759.855,Z 319.576,A -85,B 0,C 180,E1 34424.011,E2 34424.011} C_VEL
LIN {X 0,Y 759.832,Z 319.574,A -85,B 0,C 180,E1 34421.519,E2 34421.519} C_VEL
LIN {X 0,Y 759.841,Z 319.573,A -85,B 0,C 180,E1 34419.172,E2 34419.172} C_VEL
LIN {X 0,Y 759.915,Z 319.573,A -85,B 0,C 180,E1 34416.4,E2 34416.4} C_VEL
LIN {X 0,Y 759.844,Z 319.575,A -85,B 0,C 180,E1 34413.552,E2 34413.552} C_VEL
LIN {X 0,Y 759.835,Z 319.572,A -85,B 0,C 180,E1 34411.142,E2 34411.142} C_VEL
LIN {X 0,Y 759.863,Z 319.571,A -85,B 0,C 180,E1 34408.638,E2 34408.638} C_VEL
LIN {X 0,Y 759.871,Z 319.576,A -85,B 0,C 180,E1 34405.57,E2 34405.57} C_VEL
LIN {X 0,Y 759.839,Z 319.573,A -85,B 0,C 180,E1 34403.088,E2 34403.088} C_VEL
LIN {X 0,Y 759.845,Z 319.572,A -85,B 0,C 180,E1 34400.651,E2 34400.651} C_VEL
LIN {X 0,Y 759.918,Z 319.57,A -85,B 0,C 180,E1 34397.932,E2 34397.932} C_VEL
LIN {X 0,Y 759.856,Z 319.575,A -85,B 0,C 180,E1 34395.103,E2 34395.103} C_VEL
LIN {X 0,Y 759.84,Z 319.571,A -85,B 0,C 180,E1 34392.618,E2 34392.618} C_VEL
LIN {X 0,Y 759.872,Z 319.57,A -85,B 0,C 180,E1 34390.079,E2 34390.079} C_VEL
LIN {X 0,Y 759.876,Z 319.575,A -85,B 0,C 180,E1 34387.029,E2 34387.029} C_VEL
LIN {X 0,Y 759.843,Z 319.573,A -85,B 0,C 180,E1 34384.529,E2 34384.529} C_VEL
LIN {X 0,Y 759.854,Z 319.57,A -85,B 0,C 180,E1 34382.036,E2 34382.036} C_VEL
LIN {X 0,Y 759.916,Z 319.574,A -85,B 0,C 180,E1 34379.171,E2 34379.171} C_VEL
LIN {X 0,Y 759.916,Z 319.577,A -85,B 0,C 180,E1 34377.021,E2 34377.021} C_VEL
LIN {X 0,Y 758.936,Z 319.692,A -85,B 0,C 180,E1 34376.44,E2 34376.44} C_VEL
LIN {X 0,Y 752.469,Z 320.502,A -85,B 0,C 180,E1 34374.815,E2 34374.815} C_VEL
LIN {X 0,Y 751.914,Z 320.563,A -85,B 0,C 180,E1 34374.392,E2 34374.392} C_VEL
LIN {X 0,Y 751.909,Z 320.56,A -85,B 0,C 180,E1 34371.897,E2 34371.897} C_VEL
LIN {X 0,Y 751.975,Z 320.555,A -85,B 0,C 180,E1 34369.194,E2 34369.194} C_VEL
LIN {X 0,Y 751.926,Z 320.562,A -85,B 0,C 180,E1 34366.308,E2 34366.308} C_VEL
LIN {X 0,Y 751.908,Z 320.561,A -85,B 0,C 180,E1 34363.757,E2 34363.757} C_VEL
LIN {X 0,Y 751.964,Z 320.556,A -85,B 0,C 180,E1 34361.068,E2 34361.068} C_VEL
LIN {X 0,Y 751.937,Z 320.564,A -85,B 0,C 180,E1 34358.14,E2 34358.14} C_VEL
LIN {X 0,Y 751.909,Z 320.561,A -85,B 0,C 180,E1 34355.571,E2 34355.571} C_VEL
LIN {X 0,Y 751.948,Z 320.557,A -85,B 0,C 180,E1 34352.95,E2 34352.95} C_VEL
LIN {X 0,Y 751.94,Z 320.565,A -85,B 0,C 180,E1 34349.913,E2 34349.913} C_VEL
LIN {X 0,Y 751.912,Z 320.562,A -85,B 0,C 180,E1 34347.323,E2 34347.323} C_VEL
LIN {X 0,Y 751.957,Z 320.557,A -85,B 0,C 180,E1 34344.66,E2 34344.66} C_VEL
LIN {X 0,Y 751.936,Z 320.568,A -85,B 0,C 180,E1 34341.611,E2 34341.611} C_VEL
LIN {X 0,Y 751.993,Z 320.802,A -85,B 0,C 180,E1 34339.747,E2 34339.747} C_VEL
LIN {X 0,Y 753.239,Z 324.612,A -85,B 0,C 180,E1 34339.4,E2 34339.4} C_VEL
LIN {X 0,Y 753.366,Z 341.366,A -85,B 0,C 180,E1 34338.296,E2 34338.296} C_VEL
LIN {X 0,Y 753.848,Z 344.351,A -85,B 0,C 180,E1 34338.227,E2 34338.227} C_VEL
LIN {X 0,Y 753.624,Z 555.766,A -85,B 0,C 180,E1 34335.666,E2 34335.666} C_VEL
LIN {X 0,Y 753.409,Z 780.096,A -85,B 0,C 180,E1 34333.041,E2 34333.041} C_VEL
LIN {X 0,Y 753.354,Z 822.203,A -85,B 0,C 180,E1 34332.526,E2 34332.526} C_VEL
LIN {X 0,Y 753.268,Z 847.981,A -85,B 0,C 180,E1 34332.066,E2 34332.066} C_VEL
LIN {X 0,Y 753.197,Z 874.677,A -85,B 0,C 180,E1 34331.437,E2 34331.437} C_VEL
LIN {X 0,Y 753.092,Z 900.883,A -85,B 0,C 180,E1 34330.659,E2 34330.659} C_VEL
LIN {X 0,Y 752.955,Z 927.723,A -85,B 0,C 180,E1 34329.697,E2 34329.697} C_VEL
LIN {X 0,Y 752.857,Z 948.745,A -85,B 0,C 180,E1 34328.818,E2 34328.818} C_VEL
LIN {X 0,Y 752.752,Z 969.219,A -85,B 0,C 180,E1 34327.855,E2 34327.855} C_VEL
LIN {X 0,Y 752.652,Z 989.886,A -85,B 0,C 180,E1 34326.766,E2 34326.766} C_VEL
LIN {X 0,Y 752.514,Z 1014.363,A -85,B 0,C 180,E1 34325.308,E2 34325.308} C_VEL
LIN {X 0,Y 752.413,Z 1034.164,A -85,B 0,C 180,E1 34323.979,E2 34323.979} C_VEL
LIN {X 0,Y 752.322,Z 1054.427,A -85,B 0,C 180,E1 34322.475,E2 34322.475} C_VEL
LIN {X 0,Y 752.227,Z 1074.06,A -85,B 0,C 180,E1 34320.83,E2 34320.83} C_VEL
LIN {X 0,Y 752.156,Z 1089.77,A -85,B 0,C 180,E1 34319.375,E2 34319.375} C_VEL
LIN {X 0,Y 752.094,Z 1106.713,A -85,B 0,C 180,E1 34317.644,E2 34317.644} C_VEL
LIN {X 0,Y 752.037,Z 1122.344,A -85,B 0,C 180,E1 34315.825,E2 34315.825} C_VEL
LIN {X 0,Y 751.98,Z 1134.429,A -85,B 0,C 180,E1 34314.259,E2 34314.259} C_VEL
LIN {X 0,Y 751.978,Z 1145.478,A -85,B 0,C 180,E1 34312.661,E2 34312.661} C_VEL
LIN {X 0,Y 751.954,Z 1156.899,A -85,B 0,C 180,E1 34310.795,E2 34310.795} C_VEL
LIN {X 0,Y 751.918,Z 1167.362,A -85,B 0,C 180,E1 34308.771,E2 34308.771} C_VEL
LIN {X 0,Y 751.926,Z 1175.769,A -85,B 0,C 180,E1 34306.851,E2 34306.851} C_VEL
LIN {X 0,Y 751.921,Z 1183.228,A -85,B 0,C 180,E1 34304.713,E2 34304.713} C_VEL
LIN {X 0,Y 751.917,Z 1188.604,A -85,B 0,C 180,E1 34302.674,E2 34302.674} C_VEL
LIN {X 0,Y 751.91,Z 1192.332,A -85,B 0,C 180,E1 34300.652,E2 34300.652} C_VEL
LIN {X 0,Y 751.911,Z 1194.542,A -85,B 0,C 180,E1 34298.488,E2 34298.488} C_VEL
LIN {X 0,Y 751.903,Z 1194.87,A -85,B 0,C 180,E1 34296.49,E2 34296.49} C_VEL
LIN {X 0,Y 751.906,Z 1193.89,A -85,B 0,C 180,E1 34294.576,E2 34294.576} C_VEL
LIN {X 0,Y 751.909,Z 1191.027,A -85,B 0,C 180,E1 34292.439,E2 34292.439} C_VEL
LIN {X 0,Y 751.915,Z 1186.546,A -85,B 0,C 180,E1 34290.381,E2 34290.381} C_VEL
LIN {X 0,Y 751.921,Z 1180.664,A -85,B 0,C 180,E1 34288.4,E2 34288.4} C_VEL
LIN {X 0,Y 751.905,Z 1172.519,A -85,B 0,C 180,E1 34286.264,E2 34286.264} C_VEL
LIN {X 0,Y 751.935,Z 1163.091,A -85,B 0,C 180,E1 34284.277,E2 34284.277} C_VEL
LIN {X 0,Y 751.952,Z 1154.239,A -85,B 0,C 180,E1 34282.666,E2 34282.666} C_VEL
LIN {X 0,Y 751.956,Z 1144.563,A -85,B 0,C 180,E1 34281.11,E2 34281.11} C_VEL
LIN {X 0,Y 752.001,Z 1133.356,A -85,B 0,C 180,E1 34279.505,E2 34279.505} C_VEL
LIN {X 0,Y 752.062,Z 1118.77,A -85,B 0,C 180,E1 34277.64,E2 34277.64} C_VEL
LIN {X 0,Y 752.093,Z 1102.65,A -85,B 0,C 180,E1 34275.841,E2 34275.841} C_VEL
LIN {X 0,Y 752.164,Z 1087.794,A -85,B 0,C 180,E1 34274.345,E2 34274.345} C_VEL
LIN {X 0,Y 752.237,Z 1069.555,A -85,B 0,C 180,E1 34272.678,E2 34272.678} C_VEL
LIN {X 0,Y 752.334,Z 1049.742,A -85,B 0,C 180,E1 34271.078,E2 34271.078} C_VEL
LIN {X 0,Y 752.412,Z 1030.983,A -85,B 0,C 180,E1 34269.706,E2 34269.706} C_VEL
LIN {X 0,Y 752.569,Z 1007.301,A -85,B 0,C 180,E1 34268.161,E2 34268.161} C_VEL
LIN {X 0,Y 752.67,Z 986.692,A -85,B 0,C 180,E1 34266.97,E2 34266.97} C_VEL
LIN {X 0,Y 752.758,Z 966.795,A -85,B 0,C 180,E1 34265.935,E2 34265.935} C_VEL
LIN {X 0,Y 752.882,Z 943.392,A -85,B 0,C 180,E1 34264.851,E2 34264.851} C_VEL
LIN {X 0,Y 753.023,Z 917.912,A -85,B 0,C 180,E1 34263.843,E2 34263.843} C_VEL
LIN {X 0,Y 753.106,Z 896.168,A -85,B 0,C 180,E1 34263.105,E2 34263.105} C_VEL
LIN {X 0,Y 753.194,Z 873.098,A -85,B 0,C 180,E1 34262.433,E2 34262.433} C_VEL
LIN {X 0,Y 753.281,Z 846.183,A -85,B 0,C 180,E1 34261.807,E2 34261.807} C_VEL
LIN {X 0,Y 753.353,Z 819.046,A -85,B 0,C 180,E1 34261.337,E2 34261.337} C_VEL
LIN {X 0,Y 753.598,Z 576.822,A -85,B 0,C 180,E1 34258.494,E2 34258.494} C_VEL
LIN {X 0,Y 753.806,Z 365.235,A -85,B 0,C 180,E1 34255.939,E2 34255.939} C_VEL
LIN {X 0,Y 753.682,Z 342.626,A -85,B 0,C 180,E1 34255.65,E2 34255.65} C_VEL
LIN {X 0,Y 753.194,Z 340.342,A -85,B 0,C 180,E1 34255.562,E2 34255.562} C_VEL
LIN {X 0,Y 753.04,Z 323.788,A -85,B 0,C 180,E1 34254.44,E2 34254.44} C_VEL
LIN {X 0,Y 751.962,Z 320.567,A -85,B 0,C 180,E1 34254.125,E2 34254.125} C_VEL
LIN {X 0,Y 751.882,Z 320.567,A -85,B 0,C 180,E1 34251.317,E2 34251.317} C_VEL
LIN {X 0,Y 751.868,Z 320.566,A -85,B 0,C 180,E1 34249.035,E2 34249.035} C_VEL
LIN {X 0,Y 751.867,Z 320.567,A -85,B 0,C 180,E1 34246.88,E2 34246.88} C_VEL
LIN {X 0,Y 751.867,Z 320.567,A -85,B 0,C 180,E1 34244.709,E2 34244.709} C_VEL
LIN {X 0,Y 751.874,Z 320.565,A -85,B 0,C 180,E1 34242.499,E2 34242.499} C_VEL
LIN {X 0,Y 751.926,Z 320.567,A -85,B 0,C 180,E1 34239.962,E2 34239.962} C_VEL
LIN {X 0,Y 751.896,Z 320.565,A -85,B 0,C 180,E1 34237.043,E2 34237.043} C_VEL
LIN {X 0,Y 751.874,Z 320.565,A -85,B 0,C 180,E1 34234.693,E2 34234.693} C_VEL
LIN {X 0,Y 751.871,Z 320.565,A -85,B 0,C 180,E1 34232.498,E2 34232.498} C_VEL
LIN {X 0,Y 751.873,Z 320.566,A -85,B 0,C 180,E1 34230.266,E2 34230.266} C_VEL
LIN {X 0,Y 751.893,Z 320.563,A -85,B 0,C 180,E1 34227.911,E2 34227.911} C_VEL
LIN {X 0,Y 751.943,Z 320.564,A -85,B 0,C 180,E1 34225.015,E2 34225.015} C_VEL
LIN {X 0,Y 751.881,Z 320.562,A -85,B 0,C 180,E1 34222.437,E2 34222.437} C_VEL
LIN {X 0,Y 751.875,Z 320.563,A -85,B 0,C 180,E1 34220.229,E2 34220.229} C_VEL
LIN {X 0,Y 751.876,Z 320.565,A -85,B 0,C 180,E1 34217.971,E2 34217.971} C_VEL
LIN {X 0,Y 751.889,Z 320.565,A -85,B 0,C 180,E1 34215.662,E2 34215.662} C_VEL
LIN {X 0,Y 751.97,Z 320.563,A -85,B 0,C 180,E1 34212.83,E2 34212.83} C_VEL
LIN {X 0,Y 751.884,Z 320.563,A -85,B 0,C 180,E1 34210.11,E2 34210.11} C_VEL
LIN {X 0,Y 751.877,Z 320.565,A -85,B 0,C 180,E1 34207.796,E2 34207.796} C_VEL
LIN {X 0,Y 751.885,Z 320.564,A -85,B 0,C 180,E1 34205.494,E2 34205.494} C_VEL
LIN {X 0,Y 751.964,Z 320.566,A -85,B 0,C 180,E1 34202.82,E2 34202.82} C_VEL
LIN {X 0,Y 751.893,Z 320.563,A -85,B 0,C 180,E1 34199.924,E2 34199.924} C_VEL
LIN {X 0,Y 751.88,Z 320.564,A -85,B 0,C 180,E1 34197.561,E2 34197.561} C_VEL
LIN {X 0,Y 751.885,Z 320.564,A -85,B 0,C 180,E1 34195.271,E2 34195.271} C_VEL
LIN {X 0,Y 751.959,Z 320.566,A -85,B 0,C 180,E1 34192.589,E2 34192.589} C_VEL
LIN {X 0,Y 751.903,Z 320.562,A -85,B 0,C 180,E1 34189.735,E2 34189.735} C_VEL
LIN {X 0,Y 751.883,Z 320.56,A -85,B 0,C 180,E1 34187.325,E2 34187.325} C_VEL
LIN {X 0,Y 751.886,Z 320.564,A -85,B 0,C 180,E1 34185.049,E2 34185.049} C_VEL
LIN {X 0,Y 751.93,Z 320.566,A -85,B 0,C 180,E1 34182.511,E2 34182.511} C_VEL
LIN {X 0,Y 751.913,Z 320.561,A -85,B 0,C 180,E1 34179.529,E2 34179.529} C_VEL
LIN {X 0,Y 751.886,Z 320.563,A -85,B 0,C 180,E1 34177.068,E2 34177.068} C_VEL
LIN {X 0,Y 751.891,Z 320.561,A -85,B 0,C 180,E1 34174.723,E2 34174.723} C_VEL
LIN {X 0,Y 751.97,Z 320.567,A -85,B 0,C 180,E1 34171.992,E2 34171.992} C_VEL
LIN {X 0,Y 751.903,Z 320.562,A -85,B 0,C 180,E1 34169.115,E2 34169.115} C_VEL
LIN {X 0,Y 751.889,Z 320.563,A -85,B 0,C 180,E1 34166.766,E2 34166.766} C_VEL
LIN {X 0,Y 751.9,Z 320.565,A -85,B 0,C 180,E1 34164.34,E2 34164.34} C_VEL
LIN {X 0,Y 751.979,Z 320.563,A -85,B 0,C 180,E1 34161.516,E2 34161.516} C_VEL
LIN {X 0,Y 751.898,Z 320.563,A -85,B 0,C 180,E1 34158.731,E2 34158.731} C_VEL
LIN {X 0,Y 751.892,Z 320.565,A -85,B 0,C 180,E1 34156.336,E2 34156.336} C_VEL
LIN {X 0,Y 751.934,Z 320.569,A -85,B 0,C 180,E1 34153.775,E2 34153.775} C_VEL
LIN {X 0,Y 752.012,Z 320.812,A -85,B 0,C 180,E1 34153.424,E2 34153.424} C_VEL
LIN {X 0,Y 753.303,Z 324.624,A -85,B 0,C 180,E1 34153.075,E2 34153.075} C_VEL
LIN {X 0,Y 753.383,Z 351.247,A -85,B 0,C 180,E1 34151.342,E2 34151.342} C_VEL
LIN {X 0,Y 753.827,Z 354.226,A -85,B 0,C 180,E1 34151.275,E2 34151.275} C_VEL
LIN {X 0,Y 753.627,Z 564.445,A -85,B 0,C 180,E1 34148.726,E2 34148.726} C_VEL
LIN {X 0,Y 753.413,Z 790.982,A -85,B 0,C 180,E1 34146.076,E2 34146.076} C_VEL
LIN {X 0,Y 753.35,Z 832.101,A -85,B 0,C 180,E1 34145.572,E2 34145.572} C_VEL
LIN {X 0,Y 753.271,Z 858.402,A -85,B 0,C 180,E1 34145.102,E2 34145.102} C_VEL
LIN {X 0,Y 753.188,Z 885.065,A -85,B 0,C 180,E1 34144.471,E2 34144.471} C_VEL
LIN {X 0,Y 753.089,Z 911.447,A -85,B 0,C 180,E1 34143.686,E2 34143.686} C_VEL
LIN {X 0,Y 752.955,Z 937.248,A -85,B 0,C 180,E1 34142.76,E2 34142.76} C_VEL
LIN {X 0,Y 752.856,Z 958.704,A -85,B 0,C 180,E1 34141.865,E2 34141.865} C_VEL
LIN {X 0,Y 752.759,Z 977.638,A -85,B 0,C 180,E1 34140.977,E2 34140.977} C_VEL
LIN {X 0,Y 752.664,Z 997.035,A -85,B 0,C 180,E1 34139.966,E2 34139.966} C_VEL
LIN {X 0,Y 752.556,Z 1018.076,A -85,B 0,C 180,E1 34138.748,E2 34138.748} C_VEL
LIN {X 0,Y 752.411,Z 1041.012,A -85,B 0,C 180,E1 34137.246,E2 34137.246} C_VEL
LIN {X 0,Y 752.345,Z 1059.06,A -85,B 0,C 180,E1 34135.928,E2 34135.928} C_VEL
LIN {X 0,Y 752.252,Z 1077.885,A -85,B 0,C 180,E1 34134.416,E2 34134.416} C_VEL
LIN {X 0,Y 752.168,Z 1096.907,A -85,B 0,C 180,E1 34132.695,E2 34132.695} C_VEL
LIN {X 0,Y 752.092,Z 1111.836,A -85,B 0,C 180,E1 34131.199,E2 34131.199} C_VEL
LIN {X 0,Y 752.069,Z 1126.513,A -85,B 0,C 180,E1 34129.574,E2 34129.574} C_VEL
LIN {X 0,Y 752.007,Z 1142.503,A -85,B 0,C 180,E1 34127.567,E2 34127.567} C_VEL
LIN {X 0,Y 751.954,Z 1153.718,A -85,B 0,C 180,E1 34125.972,E2 34125.972} C_VEL
LIN {X 0,Y 751.955,Z 1163.592,A -85,B 0,C 180,E1 34124.398,E2 34124.398} C_VEL
LIN {X 0,Y 751.942,Z 1172.291,A -85,B 0,C 180,E1 34122.83,E2 34122.83} C_VEL
LIN {X 0,Y 751.916,Z 1180.573,A -85,B 0,C 180,E1 34121.117,E2 34121.117} C_VEL
LIN {X 0,Y 751.92,Z 1188.481,A -85,B 0,C 180,E1 34119.182,E2 34119.182} C_VEL
LIN {X 0,Y 751.915,Z 1195.351,A -85,B 0,C 180,E1 34117.027,E2 34117.027} C_VEL
LIN {X 0,Y 751.918,Z 1200.041,A -85,B 0,C 180,E1 34115.035,E2 34115.035} C_VEL
LIN {X 0,Y 751.918,Z 1203.3,A -85,B 0,C 180,E1 34112.95,E2 34112.95} C_VEL
LIN {X 0,Y 751.914,Z 1204.715,A -85,B 0,C 180,E1 34110.99,E2 34110.99} C_VEL
LIN {X 0,Y 751.891,Z 1204.827,A -85,B 0,C 180,E1 34109.39,E2 34109.39} C_VEL
LIN {X 0,Y 751.906,Z 1203.828,A -85,B 0,C 180,E1 34107.561,E2 34107.561} C_VEL
LIN {X 0,Y 751.906,Z 1200.928,A -85,B 0,C 180,E1 34105.424,E2 34105.424} C_VEL
LIN {X 0,Y 751.909,Z 1196.371,A -85,B 0,C 180,E1 34103.357,E2 34103.357} C_VEL
LIN {X 0,Y 751.92,Z 1190.361,A -85,B 0,C 180,E1 34101.358,E2 34101.358} C_VEL
LIN {X 0,Y 751.905,Z 1182.355,A -85,B 0,C 180,E1 34099.271,E2 34099.271} C_VEL
LIN {X 0,Y 751.935,Z 1173.112,A -85,B 0,C 180,E1 34097.326,E2 34097.326} C_VEL
LIN {X 0,Y 751.955,Z 1164.058,A -85,B 0,C 180,E1 34095.681,E2 34095.681} C_VEL
LIN {X 0,Y 751.954,Z 1154.214,A -85,B 0,C 180,E1 34094.103,E2 34094.103} C_VEL
LIN {X 0,Y 752.005,Z 1143.086,A -85,B 0,C 180,E1 34092.513,E2 34092.513} C_VEL
LIN {X 0,Y 752.065,Z 1127.932,A -85,B 0,C 180,E1 34090.587,E2 34090.587} C_VEL
LIN {X 0,Y 752.088,Z 1112.616,A -85,B 0,C 180,E1 34088.883,E2 34088.883} C_VEL
LIN {X 0,Y 752.166,Z 1097.976,A -85,B 0,C 180,E1 34087.408,E2 34087.408} C_VEL
LIN {X 0,Y 752.232,Z 1079.859,A -85,B 0,C 180,E1 34085.75,E2 34085.75} C_VEL
LIN {X 0,Y 752.347,Z 1060.167,A -85,B 0,C 180,E1 34084.157,E2 34084.157} C_VEL
LIN {X 0,Y 752.409,Z 1042.84,A -85,B 0,C 180,E1 34082.883,E2 34082.883} C_VEL
LIN {X 0,Y 752.521,Z 1022.27,A -85,B 0,C 180,E1 34081.511,E2 34081.511} C_VEL
LIN {X 0,Y 752.657,Z 998.639,A -85,B 0,C 180,E1 34080.121,E2 34080.121} C_VEL
LIN {X 0,Y 752.754,Z 979.254,A -85,B 0,C 180,E1 34079.103,E2 34079.103} C_VEL
LIN {X 0,Y 752.85,Z 960.434,A -85,B 0,C 180,E1 34078.213,E2 34078.213} C_VEL
LIN {X 0,Y 752.948,Z 940.603,A -85,B 0,C 180,E1 34077.375,E2 34077.375} C_VEL
LIN {X 0,Y 753.037,Z 920.043,A -85,B 0,C 180,E1 34076.609,E2 34076.609} C_VEL
LIN {X 0,Y 753.158,Z 894.913,A -85,B 0,C 180,E1 34075.802,E2 34075.802} C_VEL
LIN {X 0,Y 753.243,Z 867.449,A -85,B 0,C 180,E1 34075.094,E2 34075.094} C_VEL
LIN {X 0,Y 753.331,Z 841.93,A -85,B 0,C 180,E1 34074.586,E2 34074.586} C_VEL
LIN {X 0,Y 753.38,Z 814.81,A -85,B 0,C 180,E1 34074.197,E2 34074.197} C_VEL
LIN {X 0,Y 753.595,Z 589.429,A -85,B 0,C 180,E1 34071.57,E2 34071.57} C_VEL
LIN {X 0,Y 753.783,Z 382.952,A -85,B 0,C 180,E1 34069.078,E2 34069.078} C_VEL
LIN {X 0,Y 753.64,Z 352.252,A -85,B 0,C 180,E1 34068.688,E2 34068.688} C_VEL
LIN {X 0,Y 753.255,Z 350.376,A -85,B 0,C 180,E1 34068.621,E2 34068.621} C_VEL
LIN {X 0,Y 753.187,Z 323.923,A -85,B 0,C 180,E1 34066.87,E2 34066.87} C_VEL
LIN {X 0,Y 751.979,Z 320.565,A -85,B 0,C 180,E1 34066.553,E2 34066.553} C_VEL
LIN {X 0,Y 751.898,Z 320.566,A -85,B 0,C 180,E1 34063.775,E2 34063.775} C_VEL
LIN {X 0,Y 751.896,Z 320.563,A -85,B 0,C 180,E1 34061.371,E2 34061.371} C_VEL
LIN {X 0,Y 751.944,Z 320.561,A -85,B 0,C 180,E1 34058.778,E2 34058.778} C_VEL
LIN {X 0,Y 751.921,Z 320.565,A -85,B 0,C 180,E1 34055.793,E2 34055.793} C_VEL
LIN {X 0,Y 751.896,Z 320.563,A -85,B 0,C 180,E1 34053.314,E2 34053.314} C_VEL
LIN {X 0,Y 751.907,Z 320.559,A -85,B 0,C 180,E1 34050.884,E2 34050.884} C_VEL
LIN {X 0,Y 751.978,Z 320.563,A -85,B 0,C 180,E1 34048.08,E2 34048.08} C_VEL
LIN {X 0,Y 751.905,Z 320.564,A -85,B 0,C 180,E1 34045.269,E2 34045.269} C_VEL
LIN {X 0,Y 751.9,Z 320.559,A -85,B 0,C 180,E1 34042.849,E2 34042.849} C_VEL
LIN {X 0,Y 751.95,Z 320.558,A -85,B 0,C 180,E1 34040.226,E2 34040.226} C_VEL
LIN {X 0,Y 751.925,Z 320.563,A -85,B 0,C 180,E1 34037.25,E2 34037.25} C_VEL
LIN {X 0,Y 751.9,Z 320.562,A -85,B 0,C 180,E1 34034.714,E2 34034.714} C_VEL
LIN {X 0,Y 751.924,Z 320.557,A -85,B 0,C 180,E1 34032.206,E2 34032.206} C_VEL
LIN {X 0,Y 751.949,Z 320.565,A -85,B 0,C 180,E1 34029.182,E2 34029.182} C_VEL
LIN {X 0,Y 751.903,Z 320.56,A -85,B 0,C 180,E1 34026.567,E2 34026.567} C_VEL
LIN {X 0,Y 751.919,Z 320.56,A -85,B 0,C 180,E1 34024.041,E2 34024.041} C_VEL
LIN {X 0,Y 751.967,Z 320.564,A -85,B 0,C 180,E1 34021.067,E2 34021.067} C_VEL
LIN {X 0,Y 751.907,Z 320.563,A -85,B 0,C 180,E1 34018.4,E2 34018.4} C_VEL
LIN {X 0,Y 751.916,Z 320.557,A -85,B 0,C 180,E1 34015.882,E2 34015.882} C_VEL
LIN {X 0,Y 751.914,Z 320.563,A -85,B 0,C 180,E1 34014.392,E2 34014.392} C_VEL
LIN {X 0,Y 750.898,Z 320.689,A -85,B 0,C 180,E1 34013.805,E2 34013.805} C_VEL
LIN {X 0,Y 744.484,Z 321.487,A -85,B 0,C 180,E1 34012.161,E2 34012.161} C_VEL
LIN {X 0,Y 743.98,Z 321.548,A -85,B 0,C 180,E1 34011.733,E2 34011.733} C_VEL
LIN {X 0,Y 744.036,Z 321.552,A -85,B 0,C 180,E1 34008.811,E2 34008.811} C_VEL
LIN {X 0,Y 743.972,Z 321.548,A -85,B 0,C 180,E1 34006.079,E2 34006.079} C_VEL
LIN {X 0,Y 743.979,Z 321.548,A -85,B 0,C 180,E1 34003.526,E2 34003.526} C_VEL
LIN {X 0,Y 744.038,Z 321.55,A -85,B 0,C 180,E1 34000.614,E2 34000.614} C_VEL
LIN {X 0,Y 743.978,Z 321.552,A -85,B 0,C 180,E1 33997.894,E2 33997.894} C_VEL
LIN {X 0,Y 743.98,Z 321.547,A -85,B 0,C 180,E1 33995.293,E2 33995.293} C_VEL
LIN {X 0,Y 744.036,Z 321.55,A -85,B 0,C 180,E1 33992.465,E2 33992.465} C_VEL
LIN {X 0,Y 743.98,Z 321.552,A -85,B 0,C 180,E1 33989.646,E2 33989.646} C_VEL
LIN {X 0,Y 743.986,Z 321.549,A -85,B 0,C 180,E1 33987.023,E2 33987.023} C_VEL
LIN {X 0,Y 744.037,Z 321.553,A -85,B 0,C 180,E1 33984.128,E2 33984.128} C_VEL
LIN {X 0,Y 743.978,Z 321.557,A -85,B 0,C 180,E1 33981.321,E2 33981.321} C_VEL
LIN {X 0,Y 744.047,Z 321.631,A -85,B 0,C 180,E1 33980.258,E2 33980.258} C_VEL
LIN {X 0,Y 745.403,Z 325.127,A -85,B 0,C 180,E1 33979.918,E2 33979.918} C_VEL
LIN {X 0,Y 746.634,Z 328.545,A -85,B 0,C 180,E1 33979.596,E2 33979.596} C_VEL
LIN {X 0,Y 746.726,Z 341.353,A -85,B 0,C 180,E1 33978.746,E2 33978.746} C_VEL
LIN {X 0,Y 747.816,Z 346.118,A -85,B 0,C 180,E1 33978.612,E2 33978.612} C_VEL
LIN {X 0,Y 747.366,Z 557.298,A -85,B 0,C 180,E1 33976.033,E2 33976.033} C_VEL
LIN {X 0,Y 746.931,Z 781.407,A -85,B 0,C 180,E1 33973.389,E2 33973.389} C_VEL
LIN {X 0,Y 746.822,Z 822.785,A -85,B 0,C 180,E1 33972.877,E2 33972.877} C_VEL
LIN {X 0,Y 746.657,Z 848.816,A -85,B 0,C 180,E1 33972.405,E2 33972.405} C_VEL
LIN {X 0,Y 746.504,Z 875.252,A -85,B 0,C 180,E1 33971.775,E2 33971.775} C_VEL
LIN {X 0,Y 746.296,Z 902.532,A -85,B 0,C 180,E1 33970.956,E2 33970.956} C_VEL
LIN {X 0,Y 746.011,Z 929.074,A -85,B 0,C 180,E1 33969.985,E2 33969.985} C_VEL
LIN {X 0,Y 745.81,Z 950.908,A -85,B 0,C 180,E1 33969.057,E2 33969.057} C_VEL
LIN {X 0,Y 745.603,Z 972.11,A -85,B 0,C 180,E1 33968.038,E2 33968.038} C_VEL
LIN {X 0,Y 745.301,Z 997.49,A -85,B 0,C 180,E1 33966.652,E2 33966.652} C_VEL
LIN {X 0,Y 745.102,Z 1018.626,A -85,B 0,C 180,E1 33965.335,E2 33965.335} C_VEL
LIN {X 0,Y 744.907,Z 1039.435,A -85,B 0,C 180,E1 33963.897,E2 33963.897} C_VEL
LIN {X 0,Y 744.663,Z 1059.933,A -85,B 0,C 180,E1 33962.303,E2 33962.303} C_VEL
LIN {X 0,Y 744.528,Z 1077.582,A -85,B 0,C 180,E1 33960.774,E2 33960.774} C_VEL
LIN {X 0,Y 744.375,Z 1095.994,A -85,B 0,C 180,E1 33959.006,E2 33959.006} C_VEL
LIN {X 0,Y 744.239,Z 1111.993,A -85,B 0,C 180,E1 33957.266,E2 33957.266} C_VEL
LIN {X 0,Y 744.152,Z 1124.819,A -85,B 0,C 180,E1 33955.721,E2 33955.721} C_VEL
LIN {X 0,Y 744.075,Z 1138.089,A -85,B 0,C 180,E1 33953.942,E2 33953.942} C_VEL
LIN {X 0,Y 743.993,Z 1151.096,A -85,B 0,C 180,E1 33951.938,E2 33951.938} C_VEL
LIN {X 0,Y 743.959,Z 1160.838,A -85,B 0,C 180,E1 33950.206,E2 33950.206} C_VEL
LIN {X 0,Y 743.95,Z 1168.844,A -85,B 0,C 180,E1 33948.574,E2 33948.574} C_VEL
LIN {X 0,Y 743.933,Z 1176.377,A -85,B 0,C 180,E1 33946.796,E2 33946.796} C_VEL
LIN {X 0,Y 743.925,Z 1183.482,A -85,B 0,C 180,E1 33944.716,E2 33944.716} C_VEL
LIN {X 0,Y 743.919,Z 1188.959,A -85,B 0,C 180,E1 33942.576,E2 33942.576} C_VEL
LIN {X 0,Y 743.915,Z 1192.541,A -85,B 0,C 180,E1 33940.532,E2 33940.532} C_VEL
LIN {X 0,Y 743.914,Z 1194.579,A -85,B 0,C 180,E1 33938.424,E2 33938.424} C_VEL
LIN {X 0,Y 743.905,Z 1194.847,A -85,B 0,C 180,E1 33936.405,E2 33936.405} C_VEL
LIN {X 0,Y 743.906,Z 1193.888,A -85,B 0,C 180,E1 33934.548,E2 33934.548} C_VEL
LIN {X 0,Y 743.91,Z 1191.024,A -85,B 0,C 180,E1 33932.388,E2 33932.388} C_VEL
LIN {X 0,Y 743.916,Z 1186.541,A -85,B 0,C 180,E1 33930.308,E2 33930.308} C_VEL
LIN {X 0,Y 743.929,Z 1180.659,A -85,B 0,C 180,E1 33928.306,E2 33928.306} C_VEL
LIN {X 0,Y 743.925,Z 1172.513,A -85,B 0,C 180,E1 33926.147,E2 33926.147} C_VEL
LIN {X 0,Y 743.974,Z 1163.089,A -85,B 0,C 180,E1 33924.138,E2 33924.138} C_VEL
LIN {X 0,Y 743.984,Z 1153.786,A -85,B 0,C 180,E1 33922.432,E2 33922.432} C_VEL
LIN {X 0,Y 744.033,Z 1144.168,A -85,B 0,C 180,E1 33920.876,E2 33920.876} C_VEL
LIN {X 0,Y 744.094,Z 1132.572,A -85,B 0,C 180,E1 33919.204,E2 33919.204} C_VEL
LIN {X 0,Y 744.204,Z 1117.44,A -85,B 0,C 180,E1 33917.271,E2 33917.271} C_VEL
LIN {X 0,Y 744.317,Z 1101.911,A -85,B 0,C 180,E1 33915.531,E2 33915.531} C_VEL
LIN {X 0,Y 744.423,Z 1086.994,A -85,B 0,C 180,E1 33914.018,E2 33914.018} C_VEL
LIN {X 0,Y 744.634,Z 1067.678,A -85,B 0,C 180,E1 33912.254,E2 33912.254} C_VEL
LIN {X 0,Y 744.775,Z 1048.531,A -85,B 0,C 180,E1 33910.702,E2 33910.702} C_VEL
LIN {X 0,Y 745.012,Z 1028.136,A -85,B 0,C 180,E1 33909.208,E2 33909.208} C_VEL
LIN {X 0,Y 745.245,Z 1005.268,A -85,B 0,C 180,E1 33907.727,E2 33907.727} C_VEL
LIN {X 0,Y 745.445,Z 984.453,A -85,B 0,C 180,E1 33906.524,E2 33906.524} C_VEL
LIN {X 0,Y 745.721,Z 960.943,A -85,B 0,C 180,E1 33905.313,E2 33905.313} C_VEL
LIN {X 0,Y 745.976,Z 936.307,A -85,B 0,C 180,E1 33904.219,E2 33904.219} C_VEL
LIN {X 0,Y 746.171,Z 914.349,A -85,B 0,C 180,E1 33903.37,E2 33903.37} C_VEL
LIN {X 0,Y 746.345,Z 892.915,A -85,B 0,C 180,E1 33902.653,E2 33902.653} C_VEL
LIN {X 0,Y 746.523,Z 870.046,A -85,B 0,C 180,E1 33902.001,E2 33902.001} C_VEL
LIN {X 0,Y 746.713,Z 843.992,A -85,B 0,C 180,E1 33901.405,E2 33901.405} C_VEL
LIN {X 0,Y 746.839,Z 815.962,A -85,B 0,C 180,E1 33900.933,E2 33900.933} C_VEL
LIN {X 0,Y 747.313,Z 581.489,A -85,B 0,C 180,E1 33898.167,E2 33898.167} C_VEL
LIN {X 0,Y 747.743,Z 369.779,A -85,B 0,C 180,E1 33895.591,E2 33895.591} C_VEL
LIN {X 0,Y 747.654,Z 344.808,A -85,B 0,C 180,E1 33895.271,E2 33895.271} C_VEL
LIN {X 0,Y 746.528,Z 340.453,A -85,B 0,C 180,E1 33895.117,E2 33895.117} C_VEL
LIN {X 0,Y 746.481,Z 327.981,A -85,B 0,C 180,E1 33894.265,E2 33894.265} C_VEL
LIN {X 0,Y 744.865,Z 324.269,A -85,B 0,C 180,E1 33893.894,E2 33893.894} C_VEL
LIN {X 0,Y 743.971,Z 321.56,A -85,B 0,C 180,E1 33893.616,E2 33893.616} C_VEL
LIN {X 0,Y 743.936,Z 321.557,A -85,B 0,C 180,E1 33891.22,E2 33891.22} C_VEL
LIN {X 0,Y 743.929,Z 321.556,A -85,B 0,C 180,E1 33889.014,E2 33889.014} C_VEL
LIN {X 0,Y 743.929,Z 321.557,A -85,B 0,C 180,E1 33886.835,E2 33886.835} C_VEL
LIN {X 0,Y 743.93,Z 321.556,A -85,B 0,C 180,E1 33884.664,E2 33884.664} C_VEL
LIN {X 0,Y 743.947,Z 321.554,A -85,B 0,C 180,E1 33882.327,E2 33882.327} C_VEL
LIN {X 0,Y 744,Z 321.554,A -85,B 0,C 180,E1 33879.4,E2 33879.4} C_VEL
LIN {X 0,Y 743.937,Z 321.554,A -85,B 0,C 180,E1 33876.772,E2 33876.772} C_VEL
LIN {X 0,Y 743.932,Z 321.554,A -85,B 0,C 180,E1 33874.525,E2 33874.525} C_VEL
LIN {X 0,Y 743.937,Z 321.555,A -85,B 0,C 180,E1 33872.248,E2 33872.248} C_VEL
LIN {X 0,Y 743.997,Z 321.556,A -85,B 0,C 180,E1 33869.642,E2 33869.642} C_VEL
LIN {X 0,Y 743.959,Z 321.552,A -85,B 0,C 180,E1 33866.76,E2 33866.76} C_VEL
LIN {X 0,Y 743.937,Z 321.554,A -85,B 0,C 180,E1 33864.37,E2 33864.37} C_VEL
LIN {X 0,Y 743.936,Z 321.55,A -85,B 0,C 180,E1 33862.107,E2 33862.107} C_VEL
LIN {X 0,Y 743.947,Z 321.553,A -85,B 0,C 180,E1 33859.798,E2 33859.798} C_VEL
LIN {X 0,Y 744.032,Z 321.552,A -85,B 0,C 180,E1 33856.955,E2 33856.955} C_VEL
LIN {X 0,Y 743.946,Z 321.553,A -85,B 0,C 180,E1 33854.239,E2 33854.239} C_VEL
LIN {X 0,Y 743.938,Z 321.554,A -85,B 0,C 180,E1 33851.921,E2 33851.921} C_VEL
LIN {X 0,Y 743.946,Z 321.553,A -85,B 0,C 180,E1 33849.594,E2 33849.594} C_VEL
LIN {X 0,Y 744.042,Z 321.552,A -85,B 0,C 180,E1 33846.792,E2 33846.792} C_VEL
LIN {X 0,Y 743.952,Z 321.553,A -85,B 0,C 180,E1 33844.008,E2 33844.008} C_VEL
LIN {X 0,Y 743.941,Z 321.553,A -85,B 0,C 180,E1 33841.694,E2 33841.694} C_VEL
LIN {X 0,Y 743.946,Z 321.553,A -85,B 0,C 180,E1 33839.384,E2 33839.384} C_VEL
LIN {X 0,Y 744.02,Z 321.556,A -85,B 0,C 180,E1 33836.687,E2 33836.687} C_VEL
LIN {X 0,Y 743.962,Z 321.552,A -85,B 0,C 180,E1 33833.828,E2 33833.828} C_VEL
LIN {X 0,Y 743.944,Z 321.552,A -85,B 0,C 180,E1 33831.42,E2 33831.42} C_VEL
LIN {X 0,Y 743.946,Z 321.553,A -85,B 0,C 180,E1 33829.154,E2 33829.154} C_VEL
LIN {X 0,Y 743.987,Z 321.549,A -85,B 0,C 180,E1 33826.634,E2 33826.634} C_VEL
LIN {X 0,Y 743.97,Z 321.551,A -85,B 0,C 180,E1 33823.606,E2 33823.606} C_VEL
LIN {X 0,Y 743.947,Z 321.548,A -85,B 0,C 180,E1 33821.182,E2 33821.182} C_VEL
LIN {X 0,Y 743.95,Z 321.553,A -85,B 0,C 180,E1 33818.863,E2 33818.863} C_VEL
LIN {X 0,Y 743.996,Z 321.555,A -85,B 0,C 180,E1 33816.307,E2 33816.307} C_VEL
LIN {X 0,Y 743.972,Z 321.551,A -85,B 0,C 180,E1 33813.327,E2 33813.327} C_VEL
LIN {X 0,Y 743.949,Z 321.552,A -85,B 0,C 180,E1 33810.878,E2 33810.878} C_VEL
LIN {X 0,Y 743.959,Z 321.553,A -85,B 0,C 180,E1 33808.478,E2 33808.478} C_VEL
LIN {X 0,Y 744.036,Z 321.553,A -85,B 0,C 180,E1 33805.637,E2 33805.637} C_VEL
LIN {X 0,Y 743.958,Z 321.552,A -85,B 0,C 180,E1 33802.842,E2 33802.842} C_VEL
LIN {X 0,Y 743.952,Z 321.555,A -85,B 0,C 180,E1 33800.426,E2 33800.426} C_VEL
LIN {X 0,Y 743.994,Z 321.556,A -85,B 0,C 180,E1 33797.884,E2 33797.884} C_VEL
LIN {X 0,Y 743.982,Z 321.556,A -85,B 0,C 180,E1 33794.875,E2 33794.875} C_VEL
LIN {X 0,Y 743.985,Z 321.649,A -85,B 0,C 180,E1 33793.954,E2 33793.954} C_VEL
LIN {X 0,Y 745.069,Z 324.651,A -85,B 0,C 180,E1 33793.668,E2 33793.668} C_VEL
LIN {X 0,Y 746.726,Z 328.286,A -85,B 0,C 180,E1 33793.3,E2 33793.3} C_VEL
LIN {X 0,Y 746.775,Z 351.266,A -85,B 0,C 180,E1 33791.789,E2 33791.789} C_VEL
LIN {X 0,Y 747.796,Z 355.909,A -85,B 0,C 180,E1 33791.661,E2 33791.661} C_VEL
LIN {X 0,Y 747.37,Z 566.239,A -85,B 0,C 180,E1 33789.09,E2 33789.09} C_VEL
LIN {X 0,Y 746.935,Z 792.181,A -85,B 0,C 180,E1 33786.425,E2 33786.425} C_VEL
LIN {X 0,Y 746.818,Z 832.487,A -85,B 0,C 180,E1 33785.926,E2 33785.926} C_VEL
LIN {X 0,Y 746.66,Z 859.052,A -85,B 0,C 180,E1 33785.445,E2 33785.445} C_VEL
LIN {X 0,Y 746.493,Z 885.387,A -85,B 0,C 180,E1 33784.816,E2 33784.816} C_VEL
LIN {X 0,Y 746.294,Z 912.184,A -85,B 0,C 180,E1 33784.011,E2 33784.011} C_VEL
LIN {X 0,Y 746.013,Z 938.371,A -85,B 0,C 180,E1 33783.058,E2 33783.058} C_VEL
LIN {X 0,Y 745.813,Z 959.701,A -85,B 0,C 180,E1 33782.156,E2 33782.156} C_VEL
LIN {X 0,Y 745.618,Z 979.511,A -85,B 0,C 180,E1 33781.213,E2 33781.213} C_VEL
LIN {X 0,Y 745.411,Z 1001.051,A -85,B 0,C 180,E1 33780.066,E2 33780.066} C_VEL
LIN {X 0,Y 745.12,Z 1024.922,A -85,B 0,C 180,E1 33778.623,E2 33778.623} C_VEL
LIN {X 0,Y 744.926,Z 1043.447,A -85,B 0,C 180,E1 33777.368,E2 33777.368} C_VEL
LIN {X 0,Y 744.78,Z 1061.274,A -85,B 0,C 180,E1 33776.04,E2 33776.04} C_VEL
LIN {X 0,Y 744.532,Z 1083,A -85,B 0,C 180,E1 33774.233,E2 33774.233} C_VEL
LIN {X 0,Y 744.423,Z 1098.831,A -85,B 0,C 180,E1 33772.757,E2 33772.757} C_VEL
LIN {X 0,Y 744.288,Z 1114.958,A -85,B 0,C 180,E1 33771.102,E2 33771.102} C_VEL
LIN {X 0,Y 744.155,Z 1131.867,A -85,B 0,C 180,E1 33769.138,E2 33769.138} C_VEL
LIN {X 0,Y 744.097,Z 1144.252,A -85,B 0,C 180,E1 33767.517,E2 33767.517} C_VEL
LIN {X 0,Y 744.019,Z 1155.26,A -85,B 0,C 180,E1 33765.911,E2 33765.911} C_VEL
LIN {X 0,Y 744,Z 1165.921,A -85,B 0,C 180,E1 33764.157,E2 33764.157} C_VEL
LIN {X 0,Y 743.933,Z 1176.999,A -85,B 0,C 180,E1 33762.024,E2 33762.024} C_VEL
LIN {X 0,Y 743.93,Z 1185.541,A -85,B 0,C 180,E1 33760.062,E2 33760.062} C_VEL
LIN {X 0,Y 743.921,Z 1192.868,A -85,B 0,C 180,E1 33757.957,E2 33757.957} C_VEL
LIN {X 0,Y 743.911,Z 1198.261,A -85,B 0,C 180,E1 33755.935,E2 33755.935} C_VEL
LIN {X 0,Y 743.906,Z 1202.17,A -85,B 0,C 180,E1 33753.853,E2 33753.853} C_VEL
LIN {X 0,Y 743.906,Z 1204.381,A -85,B 0,C 180,E1 33751.771,E2 33751.771} C_VEL
LIN {X 0,Y 743.891,Z 1204.894,A -85,B 0,C 180,E1 33749.615,E2 33749.615} C_VEL
LIN {X 0,Y 743.908,Z 1203.979,A -85,B 0,C 180,E1 33747.689,E2 33747.689} C_VEL
LIN {X 0,Y 743.912,Z 1201.303,A -85,B 0,C 180,E1 33745.606,E2 33745.606} C_VEL
LIN {X 0,Y 743.919,Z 1197.153,A -85,B 0,C 180,E1 33743.595,E2 33743.595} C_VEL
LIN {X 0,Y 743.924,Z 1191.154,A -85,B 0,C 180,E1 33741.498,E2 33741.498} C_VEL
LIN {X 0,Y 743.922,Z 1183.637,A -85,B 0,C 180,E1 33739.468,E2 33739.468} C_VEL
LIN {X 0,Y 743.966,Z 1173.524,A -85,B 0,C 180,E1 33737.267,E2 33737.267} C_VEL
LIN {X 0,Y 743.999,Z 1164.525,A -85,B 0,C 180,E1 33735.604,E2 33735.604} C_VEL
LIN {X 0,Y 744.02,Z 1154.738,A -85,B 0,C 180,E1 33734.009,E2 33734.009} C_VEL
LIN {X 0,Y 744.097,Z 1144.252,A -85,B 0,C 180,E1 33732.483,E2 33732.483} C_VEL
LIN {X 0,Y 744.155,Z 1131.867,A -85,B 0,C 180,E1 33730.862,E2 33730.862} C_VEL
LIN {X 0,Y 744.287,Z 1114.958,A -85,B 0,C 180,E1 33728.898,E2 33728.898} C_VEL
LIN {X 0,Y 744.423,Z 1098.831,A -85,B 0,C 180,E1 33727.243,E2 33727.243} C_VEL
LIN {X 0,Y 744.541,Z 1082.148,A -85,B 0,C 180,E1 33725.691,E2 33725.691} C_VEL
LIN {X 0,Y 744.781,Z 1061.274,A -85,B 0,C 180,E1 33723.96,E2 33723.96} C_VEL
LIN {X 0,Y 744.926,Z 1043.446,A -85,B 0,C 180,E1 33722.632,E2 33722.632} C_VEL
LIN {X 0,Y 745.123,Z 1024.605,A -85,B 0,C 180,E1 33721.356,E2 33721.356} C_VEL
LIN {X 0,Y 745.415,Z 1000.247,A -85,B 0,C 180,E1 33719.89,E2 33719.89} C_VEL
LIN {X 0,Y 745.618,Z 979.51,A -85,B 0,C 180,E1 33718.787,E2 33718.787} C_VEL
LIN {X 0,Y 745.813,Z 959.701,A -85,B 0,C 180,E1 33717.844,E2 33717.844} C_VEL
LIN {X 0,Y 746.014,Z 938.371,A -85,B 0,C 180,E1 33716.942,E2 33716.942} C_VEL
LIN {X 0,Y 746.297,Z 911.449,A -85,B 0,C 180,E1 33715.966,E2 33715.966} C_VEL
LIN {X 0,Y 746.494,Z 885.167,A -85,B 0,C 180,E1 33715.178,E2 33715.178} C_VEL
LIN {X 0,Y 746.663,Z 858.731,A -85,B 0,C 180,E1 33714.548,E2 33714.548} C_VEL
LIN {X 0,Y 746.818,Z 832.089,A -85,B 0,C 180,E1 33714.068,E2 33714.068} C_VEL
LIN {X 0,Y 746.942,Z 789.255,A -85,B 0,C 180,E1 33713.541,E2 33713.541} C_VEL
LIN {X 0,Y 747.381,Z 562.103,A -85,B 0,C 180,E1 33710.86,E2 33710.86} C_VEL
LIN {X 0,Y 747.792,Z 355.054,A -85,B 0,C 180,E1 33708.328,E2 33708.328} C_VEL
LIN {X 0,Y 746.642,Z 350.376,A -85,B 0,C 180,E1 33708.173,E2 33708.173} C_VEL
LIN {X 0,Y 746.726,Z 328.286,A -85,B 0,C 180,E1 33706.7,E2 33706.7} C_VEL
LIN {X 0,Y 745.07,Z 324.649,A -85,B 0,C 180,E1 33706.332,E2 33706.332} C_VEL
LIN {X 0,Y 743.973,Z 321.56,A -85,B 0,C 180,E1 33706.025,E2 33706.025} C_VEL
LIN {X 0,Y 743.955,Z 321.555,A -85,B 0,C 180,E1 33703.581,E2 33703.581} C_VEL
LIN {X 0,Y 743.974,Z 321.552,A -85,B 0,C 180,E1 33701.088,E2 33701.088} C_VEL
LIN {X 0,Y 744.028,Z 321.556,A -85,B 0,C 180,E1 33698.173,E2 33698.173} C_VEL
LIN {X 0,Y 743.96,Z 321.553,A -85,B 0,C 180,E1 33695.468,E2 33695.468} C_VEL
LIN {X 0,Y 743.965,Z 321.551,A -85,B 0,C 180,E1 33693.005,E2 33693.005} C_VEL
LIN {X 0,Y 744.04,Z 321.548,A -85,B 0,C 180,E1 33690.173,E2 33690.173} C_VEL
LIN {X 0,Y 743.967,Z 321.549,A -85,B 0,C 180,E1 33687.365,E2 33687.365} C_VEL
LIN {X 0,Y 743.962,Z 321.551,A -85,B 0,C 180,E1 33684.877,E2 33684.877} C_VEL
LIN {X 0,Y 744.039,Z 321.544,A -85,B 0,C 180,E1 33682.104,E2 33682.104} C_VEL
LIN {X 0,Y 743.977,Z 321.552,A -85,B 0,C 180,E1 33679.225,E2 33679.225} C_VEL
LIN {X 0,Y 743.962,Z 321.548,A -85,B 0,C 180,E1 33676.715,E2 33676.715} C_VEL
LIN {X 0,Y 744.009,Z 321.548,A -85,B 0,C 180,E1 33674.079,E2 33674.079} C_VEL
LIN {X 0,Y 743.989,Z 321.553,A -85,B 0,C 180,E1 33671.08,E2 33671.08} C_VEL
LIN {X 0,Y 743.963,Z 321.55,A -85,B 0,C 180,E1 33668.58,E2 33668.58} C_VEL
LIN {X 0,Y 743.989,Z 321.544,A -85,B 0,C 180,E1 33666.015,E2 33666.015} C_VEL
LIN {X 0,Y 744.001,Z 321.552,A -85,B 0,C 180,E1 33662.927,E2 33662.927} C_VEL
LIN {X 0,Y 743.965,Z 321.549,A -85,B 0,C 180,E1 33660.308,E2 33660.308} C_VEL
LIN {X 0,Y 744.001,Z 321.547,A -85,B 0,C 180,E1 33657.689,E2 33657.689} C_VEL
LIN {X 0,Y 743.993,Z 321.553,A -85,B 0,C 180,E1 33654.602,E2 33654.602} C_VEL
LIN {X 0,Y 743.967,Z 321.55,A -85,B 0,C 180,E1 33652.043,E2 33652.043} C_VEL
LIN {X 0,Y 743.98,Z 321.548,A -85,B 0,C 180,E1 33651.733,E2 33651.733} C_VEL
LIN {X 0,Y 743.027,Z 321.674,A -85,B 0,C 180,E1 33651.14,E2 33651.14} C_VEL
LIN {X 0,Y 736.628,Z 322.463,A -85,B 0,C 180,E1 33649.479,E2 33649.479} C_VEL
LIN {X 0,Y 736.097,Z 322.534,A -85,B 0,C 180,E1 33649.048,E2 33649.048} C_VEL
LIN {X 0,Y 736.04,Z 322.536,A -85,B 0,C 180,E1 33646.167,E2 33646.167} C_VEL
LIN {X 0,Y 736.037,Z 322.538,A -85,B 0,C 180,E1 33643.587,E2 33643.587} C_VEL
LIN {X 0,Y 736.097,Z 322.537,A -85,B 0,C 180,E1 33640.726,E2 33640.726} C_VEL
LIN {X 0,Y 736.039,Z 322.54,A -85,B 0,C 180,E1 33637.888,E2 33637.888} C_VEL
LIN {X 0,Y 736.038,Z 322.537,A -85,B 0,C 180,E1 33635.338,E2 33635.338} C_VEL
LIN {X 0,Y 736.097,Z 322.539,A -85,B 0,C 180,E1 33632.494,E2 33632.494} C_VEL
LIN {X 0,Y 736.041,Z 322.541,A -85,B 0,C 180,E1 33629.645,E2 33629.645} C_VEL
LIN {X 0,Y 736.043,Z 322.539,A -85,B 0,C 180,E1 33627.085,E2 33627.085} C_VEL
LIN {X 0,Y 736.097,Z 322.542,A -85,B 0,C 180,E1 33624.186,E2 33624.186} C_VEL
LIN {X 0,Y 736.041,Z 322.548,A -85,B 0,C 180,E1 33621.361,E2 33621.361} C_VEL
LIN {X 0,Y 736.068,Z 322.643,A -85,B 0,C 180,E1 33620.775,E2 33620.775} C_VEL
LIN {X 0,Y 737.519,Z 326.195,A -85,B 0,C 180,E1 33620.416,E2 33620.416} C_VEL
LIN {X 0,Y 740.038,Z 332.454,A -85,B 0,C 180,E1 33619.796,E2 33619.796} C_VEL
LIN {X 0,Y 740.126,Z 341.402,A -85,B 0,C 180,E1 33619.204,E2 33619.204} C_VEL
LIN {X 0,Y 741.817,Z 348.25,A -85,B 0,C 180,E1 33618.998,E2 33618.998} C_VEL
LIN {X 0,Y 741.139,Z 558.912,A -85,B 0,C 180,E1 33616.405,E2 33616.405} C_VEL
LIN {X 0,Y 740.481,Z 783.145,A -85,B 0,C 180,E1 33613.738,E2 33613.738} C_VEL
LIN {X 0,Y 740.317,Z 823.431,A -85,B 0,C 180,E1 33613.232,E2 33613.232} C_VEL
LIN {X 0,Y 740.071,Z 849.649,A -85,B 0,C 180,E1 33612.75,E2 33612.75} C_VEL
LIN {X 0,Y 739.838,Z 875.835,A -85,B 0,C 180,E1 33612.119,E2 33612.119} C_VEL
LIN {X 0,Y 739.513,Z 903.302,A -85,B 0,C 180,E1 33611.284,E2 33611.284} C_VEL
LIN {X 0,Y 739.103,Z 928.963,A -85,B 0,C 180,E1 33610.339,E2 33610.339} C_VEL
LIN {X 0,Y 738.794,Z 951.031,A -85,B 0,C 180,E1 33609.394,E2 33609.394} C_VEL
LIN {X 0,Y 738.468,Z 974.037,A -85,B 0,C 180,E1 33608.275,E2 33608.275} C_VEL
LIN {X 0,Y 738.016,Z 999.006,A -85,B 0,C 180,E1 33606.882,E2 33606.882} C_VEL
LIN {X 0,Y 737.709,Z 1020.034,A -85,B 0,C 180,E1 33605.552,E2 33605.552} C_VEL
LIN {X 0,Y 737.394,Z 1041.926,A -85,B 0,C 180,E1 33604.009,E2 33604.009} C_VEL
LIN {X 0,Y 737.047,Z 1062.087,A -85,B 0,C 180,E1 33602.401,E2 33602.401} C_VEL
LIN {X 0,Y 736.82,Z 1081.038,A -85,B 0,C 180,E1 33600.724,E2 33600.724} C_VEL
LIN {X 0,Y 736.557,Z 1099.427,A -85,B 0,C 180,E1 33598.883,E2 33598.883} C_VEL
LIN {X 0,Y 736.397,Z 1114.236,A -85,B 0,C 180,E1 33597.23,E2 33597.23} C_VEL
LIN {X 0,Y 736.239,Z 1129.518,A -85,B 0,C 180,E1 33595.327,E2 33595.327} C_VEL
LIN {X 0,Y 736.098,Z 1143.17,A -85,B 0,C 180,E1 33593.368,E2 33593.368} C_VEL
LIN {X 0,Y 736.053,Z 1153.525,A -85,B 0,C 180,E1 33591.684,E2 33591.684} C_VEL
LIN {X 0,Y 735.99,Z 1162.547,A -85,B 0,C 180,E1 33590.02,E2 33590.02} C_VEL
LIN {X 0,Y 735.943,Z 1171.435,A -85,B 0,C 180,E1 33588.127,E2 33588.127} C_VEL
LIN {X 0,Y 735.936,Z 1179.156,A -85,B 0,C 180,E1 33586.141,E2 33586.141} C_VEL
LIN {X 0,Y 735.92,Z 1185.734,A -85,B 0,C 180,E1 33583.995,E2 33583.995} C_VEL
LIN {X 0,Y 735.913,Z 1190.534,A -85,B 0,C 180,E1 33581.839,E2 33581.839} C_VEL
LIN {X 0,Y 735.916,Z 1193.494,A -85,B 0,C 180,E1 33579.778,E2 33579.778} C_VEL
LIN {X 0,Y 735.893,Z 1194.738,A -85,B 0,C 180,E1 33577.888,E2 33577.888} C_VEL
LIN {X 0,Y 735.913,Z 1194.801,A -85,B 0,C 180,E1 33576.24,E2 33576.24} C_VEL
LIN {X 0,Y 735.907,Z 1193.728,A -85,B 0,C 180,E1 33574.364,E2 33574.364} C_VEL
LIN {X 0,Y 735.912,Z 1190.889,A -85,B 0,C 180,E1 33572.258,E2 33572.258} C_VEL
LIN {X 0,Y 735.922,Z 1186.146,A -85,B 0,C 180,E1 33570.078,E2 33570.078} C_VEL
LIN {X 0,Y 735.935,Z 1180.124,A -85,B 0,C 180,E1 33568.054,E2 33568.054} C_VEL
LIN {X 0,Y 735.956,Z 1172.168,A -85,B 0,C 180,E1 33565.949,E2 33565.949} C_VEL
LIN {X 0,Y 736.004,Z 1162.686,A -85,B 0,C 180,E1 33563.917,E2 33563.917} C_VEL
LIN {X 0,Y 736.028,Z 1153.788,A -85,B 0,C 180,E1 33562.271,E2 33562.271} C_VEL
LIN {X 0,Y 736.118,Z 1143.662,A -85,B 0,C 180,E1 33560.619,E2 33560.619} C_VEL
LIN {X 0,Y 736.231,Z 1131.108,A -85,B 0,C 180,E1 33558.802,E2 33558.802} C_VEL
LIN {X 0,Y 736.372,Z 1115.301,A -85,B 0,C 180,E1 33556.803,E2 33556.803} C_VEL
LIN {X 0,Y 736.538,Z 1100.427,A -85,B 0,C 180,E1 33555.133,E2 33555.133} C_VEL
LIN {X 0,Y 736.795,Z 1082.899,A -85,B 0,C 180,E1 33553.361,E2 33553.361} C_VEL
LIN {X 0,Y 737.028,Z 1063.343,A -85,B 0,C 180,E1 33551.614,E2 33551.614} C_VEL
LIN {X 0,Y 737.345,Z 1043.995,A -85,B 0,C 180,E1 33550.06,E2 33550.06} C_VEL
LIN {X 0,Y 737.688,Z 1021.435,A -85,B 0,C 180,E1 33548.45,E2 33548.45} C_VEL
LIN {X 0,Y 737.993,Z 1000.488,A -85,B 0,C 180,E1 33547.118,E2 33547.118} C_VEL
LIN {X 0,Y 738.433,Z 976.807,A -85,B 0,C 180,E1 33545.778,E2 33545.778} C_VEL
LIN {X 0,Y 738.781,Z 952.74,A -85,B 0,C 180,E1 33544.594,E2 33544.594} C_VEL
LIN {X 0,Y 739.083,Z 931.089,A -85,B 0,C 180,E1 33543.658,E2 33543.658} C_VEL
LIN {X 0,Y 739.418,Z 907.222,A -85,B 0,C 180,E1 33542.76,E2 33542.76} C_VEL
LIN {X 0,Y 739.782,Z 878.391,A -85,B 0,C 180,E1 33541.861,E2 33541.861} C_VEL
LIN {X 0,Y 740.069,Z 852.462,A -85,B 0,C 180,E1 33541.221,E2 33541.221} C_VEL
LIN {X 0,Y 740.284,Z 826.208,A -85,B 0,C 180,E1 33540.721,E2 33540.721} C_VEL
LIN {X 0,Y 740.446,Z 794.625,A -85,B 0,C 180,E1 33540.306,E2 33540.306} C_VEL
LIN {X 0,Y 741.093,Z 572.794,A -85,B 0,C 180,E1 33537.673,E2 33537.673} C_VEL
LIN {X 0,Y 741.769,Z 359.969,A -85,B 0,C 180,E1 33535.058,E2 33535.058} C_VEL
LIN {X 0,Y 741.66,Z 347.09,A -85,B 0,C 180,E1 33534.886,E2 33534.886} C_VEL
LIN {X 0,Y 739.907,Z 340.564,A -85,B 0,C 180,E1 33534.664,E2 33534.664} C_VEL
LIN {X 0,Y 739.83,Z 331.795,A -85,B 0,C 180,E1 33534.053,E2 33534.053} C_VEL
LIN {X 0,Y 737.086,Z 325.674,A -85,B 0,C 180,E1 33533.425,E2 33533.425} C_VEL
LIN {X 0,Y 735.99,Z 322.552,A -85,B 0,C 180,E1 33533.097,E2 33533.097} C_VEL
LIN {X 0,Y 735.99,Z 322.548,A -85,B 0,C 180,E1 33530.824,E2 33530.824} C_VEL
LIN {X 0,Y 736.001,Z 322.545,A -85,B 0,C 180,E1 33528.579,E2 33528.579} C_VEL
LIN {X 0,Y 736.087,Z 322.545,A -85,B 0,C 180,E1 33525.715,E2 33525.715} C_VEL
LIN {X 0,Y 736,Z 322.542,A -85,B 0,C 180,E1 33523,E2 33523} C_VEL
LIN {X 0,Y 735.992,Z 322.545,A -85,B 0,C 180,E1 33520.701,E2 33520.701} C_VEL
LIN {X 0,Y 735.998,Z 322.545,A -85,B 0,C 180,E1 33518.379,E2 33518.379} C_VEL
LIN {X 0,Y 736.084,Z 322.545,A -85,B 0,C 180,E1 33515.644,E2 33515.644} C_VEL
LIN {X 0,Y 736.009,Z 322.543,A -85,B 0,C 180,E1 33512.824,E2 33512.824} C_VEL
LIN {X 0,Y 735.994,Z 322.544,A -85,B 0,C 180,E1 33510.447,E2 33510.447} C_VEL
LIN {X 0,Y 735.999,Z 322.538,A -85,B 0,C 180,E1 33508.156,E2 33508.156} C_VEL
LIN {X 0,Y 736.064,Z 322.543,A -85,B 0,C 180,E1 33505.507,E2 33505.507} C_VEL
LIN {X 0,Y 736.017,Z 322.537,A -85,B 0,C 180,E1 33502.61,E2 33502.61} C_VEL
LIN {X 0,Y 735.999,Z 322.54,A -85,B 0,C 180,E1 33500.269,E2 33500.269} C_VEL
LIN {X 0,Y 736,Z 322.543,A -85,B 0,C 180,E1 33497.962,E2 33497.962} C_VEL
LIN {X 0,Y 736.025,Z 322.543,A -85,B 0,C 180,E1 33495.523,E2 33495.523} C_VEL
LIN {X 0,Y 736.026,Z 322.542,A -85,B 0,C 180,E1 33492.395,E2 33492.395} C_VEL
LIN {X 0,Y 736.001,Z 322.541,A -85,B 0,C 180,E1 33489.935,E2 33489.935} C_VEL
LIN {X 0,Y 736.004,Z 322.543,A -85,B 0,C 180,E1 33487.651,E2 33487.651} C_VEL
LIN {X 0,Y 736.051,Z 322.543,A -85,B 0,C 180,E1 33485.066,E2 33485.066} C_VEL
LIN {X 0,Y 736.027,Z 322.541,A -85,B 0,C 180,E1 33482.102,E2 33482.102} C_VEL
LIN {X 0,Y 736.004,Z 322.541,A -85,B 0,C 180,E1 33479.689,E2 33479.689} C_VEL
LIN {X 0,Y 736.007,Z 322.543,A -85,B 0,C 180,E1 33477.353,E2 33477.353} C_VEL
LIN {X 0,Y 736.076,Z 322.542,A -85,B 0,C 180,E1 33474.67,E2 33474.67} C_VEL
LIN {X 0,Y 736.019,Z 322.54,A -85,B 0,C 180,E1 33471.72,E2 33471.72} C_VEL
LIN {X 0,Y 736.005,Z 322.542,A -85,B 0,C 180,E1 33469.353,E2 33469.353} C_VEL
LIN {X 0,Y 736.015,Z 322.535,A -85,B 0,C 180,E1 33466.967,E2 33466.967} C_VEL
LIN {X 0,Y 736.096,Z 322.54,A -85,B 0,C 180,E1 33464.074,E2 33464.074} C_VEL
LIN {X 0,Y 736.012,Z 322.535,A -85,B 0,C 180,E1 33461.3,E2 33461.3} C_VEL
LIN {X 0,Y 736.009,Z 322.541,A -85,B 0,C 180,E1 33458.951,E2 33458.951} C_VEL
LIN {X 0,Y 736.034,Z 322.543,A -85,B 0,C 180,E1 33456.483,E2 33456.483} C_VEL
LIN {X 0,Y 736.038,Z 322.54,A -85,B 0,C 180,E1 33453.361,E2 33453.361} C_VEL
LIN {X 0,Y 736.011,Z 322.541,A -85,B 0,C 180,E1 33450.868,E2 33450.868} C_VEL
LIN {X 0,Y 736.021,Z 322.542,A -85,B 0,C 180,E1 33448.464,E2 33448.464} C_VEL
LIN {X 0,Y 736.095,Z 322.541,A -85,B 0,C 180,E1 33445.592,E2 33445.592} C_VEL
LIN {X 0,Y 736.018,Z 322.542,A -85,B 0,C 180,E1 33442.804,E2 33442.804} C_VEL
LIN {X 0,Y 736.014,Z 322.545,A -85,B 0,C 180,E1 33440.42,E2 33440.42} C_VEL
LIN {X 0,Y 736.075,Z 322.544,A -85,B 0,C 180,E1 33437.746,E2 33437.746} C_VEL
LIN {X 0,Y 736.039,Z 322.547,A -85,B 0,C 180,E1 33434.831,E2 33434.831} C_VEL
LIN {X 0,Y 736.045,Z 322.753,A -85,B 0,C 180,E1 33434.476,E2 33434.476} C_VEL
LIN {X 0,Y 737.281,Z 325.962,A -85,B 0,C 180,E1 33434.158,E2 33434.158} C_VEL
LIN {X 0,Y 740.205,Z 332.359,A -85,B 0,C 180,E1 33433.498,E2 33433.498} C_VEL
LIN {X 0,Y 740.195,Z 351.281,A -85,B 0,C 180,E1 33432.246,E2 33432.246} C_VEL
LIN {X 0,Y 741.797,Z 358.013,A -85,B 0,C 180,E1 33432.047,E2 33432.047} C_VEL
LIN {X 0,Y 741.142,Z 568.26,A -85,B 0,C 180,E1 33429.457,E2 33429.457} C_VEL
LIN {X 0,Y 740.483,Z 793.694,A -85,B 0,C 180,E1 33426.776,E2 33426.776} C_VEL
LIN {X 0,Y 740.313,Z 833.28,A -85,B 0,C 180,E1 33426.279,E2 33426.279} C_VEL
LIN {X 0,Y 740.075,Z 859.913,A -85,B 0,C 180,E1 33425.79,E2 33425.79} C_VEL
LIN {X 0,Y 739.822,Z 885.962,A -85,B 0,C 180,E1 33425.16,E2 33425.16} C_VEL
LIN {X 0,Y 739.516,Z 913.634,A -85,B 0,C 180,E1 33424.319,E2 33424.319} C_VEL
LIN {X 0,Y 739.092,Z 939.492,A -85,B 0,C 180,E1 33423.361,E2 33423.361} C_VEL
LIN {X 0,Y 738.79,Z 960.698,A -85,B 0,C 180,E1 33422.453,E2 33422.453} C_VEL
LIN {X 0,Y 738.49,Z 981.244,A -85,B 0,C 180,E1 33421.46,E2 33421.46} C_VEL
LIN {X 0,Y 738.11,Z 1005.698,A -85,B 0,C 180,E1 33420.125,E2 33420.125} C_VEL
LIN {X 0,Y 737.732,Z 1026.911,A -85,B 0,C 180,E1 33418.804,E2 33418.804} C_VEL
LIN {X 0,Y 737.448,Z 1045.34,A -85,B 0,C 180,E1 33417.532,E2 33417.532} C_VEL
LIN {X 0,Y 737.181,Z 1066.232,A -85,B 0,C 180,E1 33415.937,E2 33415.937} C_VEL
LIN {X 0,Y 736.85,Z 1085.147,A -85,B 0,C 180,E1 33414.305,E2 33414.305} C_VEL
LIN {X 0,Y 736.68,Z 1100.569,A -85,B 0,C 180,E1 33412.838,E2 33412.838} C_VEL
LIN {X 0,Y 736.469,Z 1117.99,A -85,B 0,C 180,E1 33411.003,E2 33411.003} C_VEL
LIN {X 0,Y 736.294,Z 1132.514,A -85,B 0,C 180,E1 33409.268,E2 33409.268} C_VEL
LIN {X 0,Y 736.197,Z 1144.254,A -85,B 0,C 180,E1 33407.711,E2 33407.711} C_VEL
LIN {X 0,Y 736.09,Z 1154.739,A -85,B 0,C 180,E1 33406.168,E2 33406.168} C_VEL
LIN {X 0,Y 736.045,Z 1164.526,A -85,B 0,C 180,E1 33404.555,E2 33404.555} C_VEL
LIN {X 0,Y 735.988,Z 1174.756,A -85,B 0,C 180,E1 33402.634,E2 33402.634} C_VEL
LIN {X 0,Y 735.948,Z 1184.913,A -85,B 0,C 180,E1 33400.331,E2 33400.331} C_VEL
LIN {X 0,Y 735.928,Z 1192.136,A -85,B 0,C 180,E1 33398.28,E2 33398.28} C_VEL
LIN {X 0,Y 735.917,Z 1197.735,A -85,B 0,C 180,E1 33396.24,E2 33396.24} C_VEL
LIN {X 0,Y 735.912,Z 1201.928,A -85,B 0,C 180,E1 33394.051,E2 33394.051} C_VEL
LIN {X 0,Y 735.912,Z 1204.213,A -85,B 0,C 180,E1 33392.024,E2 33392.024} C_VEL
LIN {X 0,Y 735.898,Z 1204.939,A -85,B 0,C 180,E1 33389.766,E2 33389.766} C_VEL
LIN {X 0,Y 735.908,Z 1203.976,A -85,B 0,C 180,E1 33387.664,E2 33387.664} C_VEL
LIN {X 0,Y 735.91,Z 1201.303,A -85,B 0,C 180,E1 33385.558,E2 33385.558} C_VEL
LIN {X 0,Y 735.92,Z 1197.152,A -85,B 0,C 180,E1 33383.525,E2 33383.525} C_VEL
LIN {X 0,Y 735.931,Z 1191.151,A -85,B 0,C 180,E1 33381.405,E2 33381.405} C_VEL
LIN {X 0,Y 735.931,Z 1183.319,A -85,B 0,C 180,E1 33379.273,E2 33379.273} C_VEL
LIN {X 0,Y 735.999,Z 1173.525,A -85,B 0,C 180,E1 33377.127,E2 33377.127} C_VEL
LIN {X 0,Y 736.045,Z 1164.526,A -85,B 0,C 180,E1 33375.445,E2 33375.445} C_VEL
LIN {X 0,Y 736.092,Z 1154.646,A -85,B 0,C 180,E1 33373.817,E2 33373.817} C_VEL
LIN {X 0,Y 736.198,Z 1143.672,A -85,B 0,C 180,E1 33372.207,E2 33372.207} C_VEL
LIN {X 0,Y 736.364,Z 1129.29,A -85,B 0,C 180,E1 33370.322,E2 33370.322} C_VEL
LIN {X 0,Y 736.522,Z 1112.62,A -85,B 0,C 180,E1 33368.414,E2 33368.414} C_VEL
LIN {X 0,Y 736.685,Z 1097.979,A -85,B 0,C 180,E1 33366.906,E2 33366.906} C_VEL
LIN {X 0,Y 736.985,Z 1079.52,A -85,B 0,C 180,E1 33365.184,E2 33365.184} C_VEL
LIN {X 0,Y 737.229,Z 1060.167,A -85,B 0,C 180,E1 33363.587,E2 33363.587} C_VEL
LIN {X 0,Y 737.478,Z 1042.501,A -85,B 0,C 180,E1 33362.263,E2 33362.263} C_VEL
LIN {X 0,Y 737.895,Z 1020.413,A -85,B 0,C 180,E1 33360.77,E2 33360.77} C_VEL
LIN {X 0,Y 738.221,Z 997.841,A -85,B 0,C 180,E1 33359.431,E2 33359.431} C_VEL
LIN {X 0,Y 738.518,Z 977.732,A -85,B 0,C 180,E1 33358.362,E2 33358.362} C_VEL
LIN {X 0,Y 738.84,Z 956.624,A -85,B 0,C 180,E1 33357.361,E2 33357.361} C_VEL
LIN {X 0,Y 739.293,Z 929.68,A -85,B 0,C 180,E1 33356.257,E2 33356.257} C_VEL
LIN {X 0,Y 739.567,Z 907.054,A -85,B 0,C 180,E1 33355.472,E2 33355.472} C_VEL
LIN {X 0,Y 739.849,Z 883.683,A -85,B 0,C 180,E1 33354.78,E2 33354.78} C_VEL
LIN {X 0,Y 740.113,Z 856.978,A -85,B 0,C 180,E1 33354.148,E2 33354.148} C_VEL
LIN {X 0,Y 740.323,Z 829.711,A -85,B 0,C 180,E1 33353.667,E2 33353.667} C_VEL
LIN {X 0,Y 740.657,Z 731.552,A -85,B 0,C 180,E1 33352.493,E2 33352.493} C_VEL
LIN {X 0,Y 741.332,Z 508.633,A -85,B 0,C 180,E1 33349.818,E2 33349.818} C_VEL
LIN {X 0,Y 741.675,Z 356.755,A -85,B 0,C 180,E1 33347.928,E2 33347.928} C_VEL
LIN {X 0,Y 740.053,Z 350.376,A -85,B 0,C 180,E1 33347.714,E2 33347.714} C_VEL
LIN {X 0,Y 740.205,Z 332.359,A -85,B 0,C 180,E1 33346.502,E2 33346.502} C_VEL
LIN {X 0,Y 736.096,Z 323.053,A -85,B 0,C 180,E1 33345.549,E2 33345.549} C_VEL
LIN {X 0,Y 736.018,Z 322.549,A -85,B 0,C 180,E1 33345.495,E2 33345.495} C_VEL
LIN {X 0,Y 736.077,Z 322.542,A -85,B 0,C 180,E1 33342.818,E2 33342.818} C_VEL
LIN {X 0,Y 736.038,Z 322.545,A -85,B 0,C 180,E1 33339.869,E2 33339.869} C_VEL
LIN {X 0,Y 736.018,Z 322.542,A -85,B 0,C 180,E1 33337.373,E2 33337.373} C_VEL
LIN {X 0,Y 736.041,Z 322.54,A -85,B 0,C 180,E1 33334.866,E2 33334.866} C_VEL
LIN {X 0,Y 736.06,Z 322.538,A -85,B 0,C 180,E1 33331.808,E2 33331.808} C_VEL
LIN {X 0,Y 736.022,Z 322.542,A -85,B 0,C 180,E1 33329.279,E2 33329.279} C_VEL
LIN {X 0,Y 736.028,Z 322.533,A -85,B 0,C 180,E1 33326.809,E2 33326.809} C_VEL
